  MoveL 4571 to (30.32, 60.2, -219.61) mm, rotated rx -167.81 ry 3.47 rz -52.11 deg; joints [-1.862, -33.382, 100.556, 145.163, 95.8, 28.312, -1.714]
  MoveL 4572 to (32.46, 60.06, -219.75) mm, rotated rx -167.81 ry 3.47 rz -52.11 deg; joints [-1.941, -33.35, 100.546, 145.092, 95.836, 28.324, -1.714]
  MoveL 4573 to (34.58, 59.96, -219.77) mm, rotated rx -167.81 ry 3.47 rz -52.11 deg; joints [-2.017, -33.309, 100.528, 145.023, 95.871, 28.336, -1.714]
  MoveL 4574 to (35.08, 59.57, -220.44) mm, rotated rx -167.81 ry 3.47 rz -52.11 deg; joints [-2.042, -33.346, 100.585, 144.999, 95.893, 28.332, -1.714]
  MoveL 4575 to (34.76, 59.5, -220.77) mm, rotated rx -167.81 ry 3.47 rz -52.11 deg; joints [-2.034, -33.375, 100.611, 145.006, 95.89, 28.331, -1.714]
  MoveL 4576 to (34.71, 59.48, -220.97) mm, rotated rx -167.81 ry 3.47 rz -52.11 deg; joints [-2.035, -33.389, 100.623, 145.005, 95.888, 28.332, -1.714]
  MoveL 4577 to (34.93, 59.52, -221.07) mm, rotated rx -167.81 ry 3.47 rz -52.11 deg; joints [-2.044, -33.39, 100.622, 144.997, 95.888, 28.337, -1.714]
  MoveL 4578 to (35.33, 59.66, -221.1) mm, rotated rx -167.81 ry 3.47 rz -52.11 deg; joints [-2.059, -33.381, 100.607, 144.985, 95.886, 28.345, -1.714]
  MoveC 4579 to (36.23, 60.13, -221.1) mm, rotated rx -167.81 ry 3.47 rz -52.11 deg; joints [-2.092, -33.356, 100.556, 144.957, 95.873, 28.37, -1.714] to (37.1, 60.66, -221.1) mm, rotated rx -167.81 ry 3.47 rz -52.11 deg; joints [-2.124, -33.33, 100.502, 144.93, 95.857, 28.397, -1.714]
  MoveL 4580 to (37.1, 60.66, -221.1) mm, rotated rx -167.81 ry 3.47 rz -52.11 deg; joints [-2.124, -33.331, 100.502, 144.93, 95.856, 28.397, -1.714]
  MoveL 4581 to (37.57, 60.93, -221.12) mm, rotated rx -167.81 ry 3.47 rz -52.11 deg; joints [-2.142, -33.318, 100.475, 144.915, 95.848, 28.411, -1.714]
  MoveL 4582 to (38.04, 61.18, -221.17) mm, rotated rx -167.81 ry 3.47 rz -52.11 deg; joints [-2.16, -33.308, 100.45, 144.9, 95.84, 28.425, -1.714]
  MoveL 4583 to (38.56, 61.45, -221.24) mm, rotated rx -167.81 ry 3.47 rz -52.11 deg; joints [-2.179, -33.298, 100.425, 144.883, 95.833, 28.44, -1.714]
  MoveL 4584 to (39.08, 61.73, -221.28) mm, rotated rx -167.81 ry 3.47 rz -52.11 deg; joints [-2.199, -33.285, 100.397, 144.867, 95.824, 28.456, -1.714]
  MoveL 4585 to (40.13, 62.35, -221.3) mm, rotated rx -167.81 ry 3.47 rz -52.11 deg; joints [-2.238, -33.256, 100.333, 144.835, 95.805, 28.488, -1.714]
  MoveL 4586 to (40.62, 62.62, -221.34) mm, rotated rx -167.81 ry 3.47 rz -52.11 deg; joints [-2.256, -33.244, 100.307, 144.819, 95.797, 28.502, -1.714]
  MoveL 4587 to (41.05, 62.82, -221.41) mm, rotated rx -167.81 ry 3.47 rz -52.11 deg; joints [-2.272, -33.237, 100.288, 144.805, 95.791, 28.514, -1.714]
  MoveL 4588 to (41.45, 63, -221.5) mm, rotated rx -167.81 ry 3.47 rz -52.11 deg; joints [-2.288, -33.232, 100.272, 144.792, 95.786, 28.525, -1.714]
  MoveL 4589 to (41.83, 63.19, -221.56) mm, rotated rx -167.81 ry 3.47 rz -52.11 deg; joints [-2.303, -33.225, 100.255, 144.78, 95.78, 28.536, -1.714]
  MoveL 4590 to (42.22, 63.4, -221.6) mm, rotated rx -167.81 ry 3.47 rz -52.11 deg; joints [-2.317, -33.216, 100.234, 144.767, 95.774, 28.548, -1.714]
  MoveL 4591 to (44.46, 64.76, -221.6) mm, rotated rx -167.81 ry 3.47 rz -52.11 deg; joints [-2.399, -33.15, 100.092, 144.699, 95.731, 28.618, -1.714]
  MoveL 4592 to (47.08, 66.03, -221.94) mm, rotated rx -167.81 ry 3.47 rz -52.11 deg; joints [-2.498, -33.098, 99.968, 144.615, 95.694, 28.692, -1.714]
  MoveL 4593 to (48.31, 66.38, -222.37) mm, rotated rx -167.81 ry 3.47 rz -52.11 deg; joints [-2.548, -33.094, 99.943, 144.572, 95.688, 28.72, -1.714]
  MoveL 4594 to (49.5, 66.55, -222.98) mm, rotated rx -167.81 ry 3.47 rz -52.11 deg; joints [-2.598, -33.105, 99.942, 144.529, 95.691, 28.743, -1.714]
  MoveL 4595 to (50.63, 66.52, -223.75) mm, rotated rx -167.81 ry 3.47 rz -52.11 deg; joints [-2.648, -33.13, 99.966, 144.484, 95.701, 28.76, -1.714]
  MoveL 4596 to (51.72, 66.31, -224.7) mm, rotated rx -167.81 ry 3.47 rz -52.11 deg; joints [-2.698, -33.17, 100.014, 144.439, 95.719, 28.771, -1.714]
  MoveL 4597 to (53.75, 65.31, -227.12) mm, rotated rx -167.81 ry 3.47 rz -52.11 deg; joints [-2.799, -33.293, 100.184, 144.347, 95.78, 28.776, -1.714]
  MoveL 4598 to (55.07, 63.94, -229.53) mm, rotated rx -167.81 ry 3.47 rz -52.11 deg; joints [-2.875, -33.436, 100.393, 144.276, 95.851, 28.762, -1.714]
  MoveL 4599 to (55.28, 63.26, -230.48) mm, rotated rx -167.81 ry 3.47 rz -52.11 deg; joints [-2.893, -33.501, 100.491, 144.257, 95.882, 28.748, -1.714]
  MoveL 4600 to (55.19, 62.59, -231.25) mm, rotated rx -167.81 ry 3.47 rz -52.11 deg; joints [-2.899, -33.561, 100.584, 144.25, 95.91, 28.731, -1.714]
  MoveL 4601 to (55.03, 62.26, -231.58) mm, rotated rx -167.81 ry 3.47 rz -52.11 deg; joints [-2.897, -33.59, 100.629, 144.251, 95.923, 28.72, -1.714]
  MoveL 4602 to (54.8, 61.92, -231.86) mm, rotated rx -167.81 ry 3.47 rz -52.11 deg; joints [-2.892, -33.617, 100.673, 144.255, 95.936, 28.709, -1.714]
  MoveL 4603 to (54.11, 61.26, -232.29) mm, rotated rx -167.81 ry 3.47 rz -52.11 deg; joints [-2.871, -33.668, 100.758, 144.271, 95.958, 28.683, -1.714]
  MoveL 4604 to (53.11, 60.6, -232.55) mm, rotated rx -167.81 ry 3.47 rz -52.11 deg; joints [-2.838, -33.715, 100.838, 144.298, 95.978, 28.652, -1.714]
  MoveL 4605 to (51.82, 59.94, -232.63) mm, rotated rx -167.81 ry 3.47 rz -52.11 deg; joints [-2.792, -33.757, 100.915, 144.337, 95.995, 28.618, -1.714]
  MoveL 4606 to (51.34, 59.73, -232.63) mm, rotated rx -167.81 ry 3.47 rz -52.11 deg; joints [-2.775, -33.77, 100.939, 144.352, 96, 28.606, -1.714]
  MoveL 4607 to (50.92, 59.56, -232.6) mm, rotated rx -167.81 ry 3.47 rz -52.11 deg; joints [-2.759, -33.779, 100.957, 144.365, 96.004, 28.596, -1.714]
  MoveL 4608 to (50.53, 59.42, -232.55) mm, rotated rx -167.81 ry 3.47 rz -52.11 deg; joints [-2.744, -33.786, 100.971, 144.378, 96.007, 28.586, -1.714]
  MoveL 4609 to (50.14, 59.29, -232.48) mm, rotated rx -167.81 ry 3.47 rz -52.11 deg; joints [-2.729, -33.792, 100.984, 144.391, 96.009, 28.578, -1.714]
  MoveL 4610 to (49.72, 59.14, -232.43) mm, rotated rx -167.81 ry 3.47 rz -52.11 deg; joints [-2.714, -33.8, 101, 144.404, 96.012, 28.568, -1.714]
  MoveL 4611 to (49.26, 58.94, -232.41) mm, rotated rx -167.81 ry 3.47 rz -52.11 deg; joints [-2.696, -33.811, 101.021, 144.419, 96.017, 28.556, -1.714]
  MoveL 4612 to (44.04, 56.58, -232.4) mm, rotated rx -167.81 ry 3.47 rz -52.11 deg; joints [-2.506, -33.953, 101.285, 144.581, 96.072, 28.425, -1.714]
  MoveL 4613 to (43.33, 56.28, -232.39) mm, rotated rx -167.81 ry 3.47 rz -52.11 deg; joints [-2.48, -33.971, 101.318, 144.603, 96.079, 28.408, -1.714]
  MoveL 4614 to (42.72, 56.05, -232.38) mm, rotated rx -167.81 ry 3.47 rz -52.11 deg; joints [-2.457, -33.987, 101.345, 144.622, 96.083, 28.395, -1.714]
  MoveL 4615 to (42.16, 55.93, -232.37) mm, rotated rx -167.81 ry 3.47 rz -52.11 deg; joints [-2.437, -34, 101.362, 144.64, 96.082, 28.386, -1.714]
  MoveL 4616 to (41.62, 55.89, -232.33) mm, rotated rx -167.81 ry 3.47 rz -52.11 deg; joints [-2.417, -34.009, 101.371, 144.658, 96.077, 28.38, -1.714]
  MoveL 4617 to (41.29, 55.92, -232.17) mm, rotated rx -167.81 ry 3.47 rz -52.11 deg; joints [-2.403, -34.005, 101.365, 144.67, 96.072, 28.377, -1.714]
  MoveL 4618 to (41.29, 55.95, -231.86) mm, rotated rx -167.81 ry 3.47 rz -52.11 deg; joints [-2.399, -33.985, 101.348, 144.673, 96.074, 28.374, -1.714]
  MoveL 4619 to (41.65, 55.96, -231.37) mm, rotated rx -167.81 ry 3.47 rz -52.11 deg; joints [-2.407, -33.947, 101.319, 144.667, 96.083, 28.371, -1.714]
  MoveL 4620 to (41.42, 56.54, -230.4) mm, rotated rx -167.81 ry 3.47 rz -52.11 deg; joints [-2.387, -33.883, 101.228, 144.685, 96.057, 28.38, -1.714]
  MoveL 4621 to (39.59, 56.9, -230.1) mm, rotated rx -167.81 ry 3.47 rz -52.11 deg; joints [-2.318, -33.897, 101.21, 144.749, 96.015, 28.377, -1.714]
  MoveL 4622 to (37.66, 57.25, -229.89) mm, rotated rx -167.81 ry 3.47 rz -52.11 deg; joints [-2.246, -33.919, 101.196, 144.815, 95.971, 28.374, -1.714]
  MoveL 4623 to (35.56, 57.62, -229.77) mm, rotated rx -167.81 ry 3.47 rz -52.11 deg; joints [-2.17, -33.948, 101.188, 144.885, 95.922, 28.372, -1.714]
  MoveL 4624 to (31.35, 58.33, -229.77) mm, rotated rx -167.81 ry 3.47 rz -52.11 deg; joints [-2.019, -34.024, 101.185, 145.024, 95.824, 28.37, -1.714]
  MoveL 4625 to (29.4, 58.66, -229.68) mm, rotated rx -167.81 ry 3.47 rz -52.11 deg; joints [-1.948, -34.054, 101.179, 145.089, 95.779, 28.367, -1.714]
  MoveL 4626 to (27.29, 59.01, -229.68) mm, rotated rx -167.81 ry 3.47 rz -52.11 deg; joints [-1.873, -34.092, 101.177, 145.158, 95.73, 28.366, -1.714]
  MoveL 4627 to (25.18, 59.46, -229.68) mm, rotated rx -167.81 ry 3.47 rz -52.11 deg; joints [-1.797, -34.128, 101.166, 145.228, 95.675, 28.369, -1.714]
  MoveL 4628 to (22.7, 60.03, -229.5) mm, rotated rx -167.81 ry 3.47 rz -52.11 deg; joints [-1.707, -34.158, 101.142, 145.312, 95.609, 28.371, -1.714]
  MoveL 4629 to (20.49, 60.27, -229.27) mm, rotated rx -167.81 ry 3.47 rz -52.11 deg; joints [-1.625, -34.185, 101.138, 145.386, 95.566, 28.362, -1.714]
  MoveL 4630 to (18.33, 60.54, -229.15) mm, rotated rx -167.81 ry 3.47 rz -52.11 deg; joints [-1.546, -34.217, 101.137, 145.458, 95.521, 28.355, -1.714]
  MoveL 4631 to (16.23, 60.89, -229.04) mm, rotated rx -167.81 ry 3.47 rz -52.11 deg; joints [-1.469, -34.247, 101.128, 145.528, 95.472, 28.352, -1.714]
  MoveL 4632 to (14.12, 61.23, -228.82) mm, rotated rx -167.81 ry 3.47 rz -52.11 deg; joints [-1.392, -34.271, 101.115, 145.599, 95.424, 28.348, -1.714]
  MoveL 4633 to (12.02, 61.58, -228.72) mm, rotated rx -167.81 ry 3.47 rz -52.11 deg; joints [-1.315, -34.301, 101.106, 145.669, 95.375, 28.345, -1.714]
  MoveL 4634 to (9.91, 61.92, -228.61) mm, rotated rx -167.81 ry 3.47 rz -52.11 deg; joints [-1.239, -34.331, 101.097, 145.739, 95.326, 28.342, -1.714]
  MoveL 4635 to (7.8, 62.25, -228.39) mm, rotated rx -167.81 ry 3.47 rz -52.11 deg; joints [-1.161, -34.354, 101.084, 145.81, 95.278, 28.338, -1.714]
  MoveL 4636 to (5.7, 62.59, -228.29) mm, rotated rx -167.81 ry 3.47 rz -52.11 deg; joints [-1.085, -34.384, 101.075, 145.88, 95.229, 28.335, -1.714]
  MoveL 4637 to (3.59, 62.93, -228.18) mm, rotated rx -167.81 ry 3.47 rz -52.11 deg; joints [-1.008, -34.414, 101.065, 145.95, 95.18, 28.332, -1.714]
  MoveL 4638 to (1.48, 63.24, -227.98) mm, rotated rx -167.81 ry 3.47 rz -52.11 deg; joints [-0.93, -34.438, 101.053, 146.021, 95.132, 28.326, -1.714]
  MoveL 4639 to (-0.63, 63.58, -227.88) mm, rotated rx -167.81 ry 3.47 rz -52.11 deg; joints [-0.854, -34.468, 101.044, 146.091, 95.083, 28.323, -1.714]
  MoveL 4640 to (-2.46, 63.79, -227.62) mm, rotated rx -167.81 ry 3.47 rz -52.11 deg; joints [-0.785, -34.485, 101.033, 146.153, 95.045, 28.315, -1.714]
  MoveL 4641 to (-4.13, 63.93, -227.25) mm, rotated rx -167.81 ry 3.47 rz -52.11 deg; joints [-0.721, -34.492, 101.022, 146.211, 95.016, 28.304, -1.714]
  MoveL 4642 to (-5.65, 63.98, -226.75) mm, rotated rx -167.81 ry 3.47 rz -52.11 deg; joints [-0.661, -34.49, 101.01, 146.265, 94.994, 28.29, -1.714]
  MoveL 4643 to (-4.6, 63.55, -225.91) mm, rotated rx -167.81 ry 3.47 rz -52.11 deg; joints [-0.688, -34.423, 100.994, 146.239, 95.042, 28.27, -1.714]
  MoveL 4644 to (-4.93, 63.61, -225.88) mm, rotated rx -167.81 ry 3.47 rz -52.11 deg; joints [-0.676, -34.427, 100.991, 146.25, 95.034, 28.27, -1.714]
  MoveL 4645 to (-5.24, 63.69, -225.83) mm, rotated rx -167.81 ry 3.47 rz -52.11 deg; joints [-0.664, -34.429, 100.985, 146.26, 95.025, 28.271, -1.714]
  MoveL 4646 to (-5.56, 63.87, -225.78) mm, rotated rx -167.81 ry 3.47 rz -52.11 deg; joints [-0.652, -34.429, 100.972, 146.272, 95.011, 28.274, -1.714]
  MoveL 4647 to (-5.9, 64.11, -225.74) mm, rotated rx -167.81 ry 3.47 rz -52.11 deg; joints [-0.64, -34.43, 100.954, 146.283, 94.993, 28.28, -1.714]
  MoveL 4648 to (-6.28, 64.42, -225.72) mm, rotated rx -167.81 ry 3.47 rz -52.11 deg; joints [-0.627, -34.431, 100.932, 146.296, 94.971, 28.289, -1.714]
  MoveL 4649 to (-9.71, 67.65, -225.72) mm, rotated rx -167.81 ry 3.47 rz -52.11 deg; joints [-0.511, -34.447, 100.701, 146.41, 94.74, 28.388, -1.714]
  MoveL 4650 to (-10.01, 67.91, -225.69) mm, rotated rx -167.81 ry 3.47 rz -52.11 deg; joints [-0.501, -34.447, 100.682, 146.421, 94.721, 28.395, -1.714]
  MoveL 4651 to (-10.39, 68.27, -225.69) mm, rotated rx -167.81 ry 3.47 rz -52.11 deg; joints [-0.488, -34.449, 100.656, 146.433, 94.695, 28.406, -1.714]
  MoveL 4652 to (-11.16, 68.96, -225.65) mm, rotated rx -167.81 ry 3.47 rz -52.11 deg; joints [-0.461, -34.45, 100.605, 146.459, 94.646, 28.426, -1.714]
  MoveL 4653 to (-13.06, 70.76, -225.65) mm, rotated rx -167.81 ry 3.47 rz -52.11 deg; joints [-0.397, -34.459, 100.476, 146.522, 94.517, 28.48, -1.714]
  MoveL 4654 to (-13.85, 71.42, -225.63) mm, rotated rx -167.81 ry 3.47 rz -52.11 deg; joints [-0.371, -34.462, 100.429, 146.548, 94.468, 28.5, -1.714]
  MoveL 4655 to (-14.92, 72.4, -225.7) mm, rotated rx -167.81 ry 3.47 rz -52.11 deg; joints [-0.336, -34.471, 100.361, 146.582, 94.397, 28.53, -1.714]
  MoveL 4656 to (-15.68, 73.29, -225.95) mm, rotated rx -167.81 ry 3.47 rz -52.11 deg; joints [-0.314, -34.487, 100.307, 146.605, 94.333, 28.561, -1.714]
  MoveL 4657 to (-16.13, 74.1, -226.39) mm, rotated rx -167.81 ry 3.47 rz -52.11 deg; joints [-0.304, -34.51, 100.266, 146.616, 94.277, 28.593, -1.714]
  MoveL 4658 to (-16.25, 74.47, -226.68) mm, rotated rx -167.81 ry 3.47 rz -52.11 deg; joints [-0.305, -34.525, 100.25, 146.617, 94.252, 28.61, -1.714]
  MoveL 4659 to (-16.28, 74.82, -227.02) mm, rotated rx -167.81 ry 3.47 rz -52.11 deg; joints [-0.308, -34.541, 100.237, 146.615, 94.229, 28.627, -1.714]
  MoveL 4660 to (-16.13, 75.46, -227.83) mm, rotated rx -167.81 ry 3.47 rz -52.11 deg; joints [-0.324, -34.578, 100.221, 146.602, 94.188, 28.662, -1.714]
  MoveL 4661 to (-15.68, 76.02, -228.83) mm, rotated rx -167.81 ry 3.47 rz -52.11 deg; joints [-0.354, -34.623, 100.219, 146.578, 94.155, 28.698, -1.714]
  MoveL 4662 to (-13.85, 76.87, -231.39) mm, rotated rx -167.81 ry 3.47 rz -52.11 deg; joints [-0.451, -34.733, 100.251, 146.496, 94.112, 28.775, -1.714]
  MoveL 4663 to (-11.47, 77.17, -233.95) mm, rotated rx -167.81 ry 3.47 rz -52.11 deg; joints [-0.567, -34.843, 100.324, 146.395, 94.109, 28.835, -1.714]
  MoveL 4664 to (-9.19, 76.69, -235.78) mm, rotated rx -167.81 ry 3.47 rz -52.11 deg; joints [-0.668, -34.921, 100.428, 146.303, 94.153, 28.857, -1.714]
  MoveL 4665 to (-8.08, 76.15, -236.42) mm, rotated rx -167.81 ry 3.47 rz -52.11 deg; joints [-0.714, -34.948, 100.491, 146.261, 94.193, 28.852, -1.714]
  MoveL 4666 to (-7, 75.42, -236.88) mm, rotated rx -167.81 ry 3.47 rz -52.11 deg; joints [-0.757, -34.968, 100.562, 146.222, 94.246, 28.838, -1.714]
  MoveL 4667 to (-4.92, 73.38, -237.25) mm, rotated rx -167.81 ry 3.47 rz -52.11 deg; joints [-0.831, -34.984, 100.727, 146.149, 94.387, 28.781, -1.714]
  MoveL 4668 to (-2.9, 70.96, -237.25) mm, rotated rx -167.81 ry 3.47 rz -52.11 deg; joints [-0.899, -34.983, 100.905, 146.082, 94.55, 28.704, -1.714]
  MoveL 4669 to (-2.23, 70.2, -237.26) mm, rotated rx -167.81 ry 3.47 rz -52.11 deg; joints [-0.921, -34.983, 100.962, 146.059, 94.603, 28.68, -1.714]
  MoveL 4670 to (-1.56, 69.4, -237.26) mm, rotated rx -167.81 ry 3.47 rz -52.11 deg; joints [-0.944, -34.983, 101.021, 146.037, 94.657, 28.654, -1.714]
  MoveL 4671 to (-1.24, 69.02, -237.27) mm, rotated rx -167.81 ry 3.47 rz -52.11 deg; joints [-0.955, -34.983, 101.049, 146.026, 94.683, 28.642, -1.714]
  MoveL 4672 to (-0.8, 68.52, -237.3) mm, rotated rx -167.81 ry 3.47 rz -52.11 deg; joints [-0.969, -34.984, 101.087, 146.011, 94.716, 28.627, -1.714]
  MoveL 4673 to (-0.4, 68.08, -237.35) mm, rotated rx -167.81 ry 3.47 rz -52.11 deg; joints [-0.984, -34.987, 101.121, 145.997, 94.746, 28.613, -1.714]
  MoveL 4674 to (-0.04, 67.72, -237.43) mm, rotated rx -167.81 ry 3.47 rz -52.11 deg; joints [-0.997, -34.99, 101.15, 145.984, 94.77, 28.603, -1.714]
  MoveL 4675 to (0.28, 67.39, -237.48) mm, rotated rx -167.81 ry 3.47 rz -52.11 deg; joints [-1.008, -34.992, 101.177, 145.973, 94.793, 28.594, -1.714]
  MoveL 4676 to (0.6, 67.04, -237.51) mm, rotated rx -167.81 ry 3.47 rz -52.11 deg; joints [-1.019, -34.993, 101.203, 145.962, 94.816, 28.583, -1.714]
  MoveL 4677 to (1.6, 65.84, -237.51) mm, rotated rx -167.81 ry 3.47 rz -52.11 deg; joints [-1.053, -34.992, 101.291, 145.928, 94.898, 28.545, -1.714]
  MoveL 4678 to (1.94, 65.47, -237.53) mm, rotated rx -167.81 ry 3.47 rz -52.11 deg; joints [-1.065, -34.992, 101.319, 145.916, 94.923, 28.533, -1.714]
  MoveL 4679 to (2.25, 65.16, -237.55) mm, rotated rx -167.81 ry 3.47 rz -52.11 deg; joints [-1.076, -34.993, 101.342, 145.905, 94.945, 28.524, -1.714]
  MoveL 4680 to (2.55, 64.91, -237.6) mm, rotated rx -167.81 ry 3.47 rz -52.11 deg; joints [-1.086, -34.994, 101.361, 145.895, 94.962, 28.517, -1.714]
  MoveL 4681 to (2.81, 64.76, -237.67) mm, rotated rx -167.81 ry 3.47 rz -52.11 deg; joints [-1.096, -34.995, 101.373, 145.885, 94.974, 28.514, -1.714]
  MoveL 4682 to (3.07, 64.67, -237.74) mm, rotated rx -167.81 ry 3.47 rz -52.11 deg; joints [-1.106, -34.996, 101.381, 145.876, 94.982, 28.513, -1.714]
  MoveL 4683 to (1.89, 65.73, -238.54) mm, rotated rx -167.81 ry 3.47 rz -52.11 deg; joints [-1.075, -35.053, 101.345, 145.908, 94.898, 28.555, -1.714]
  MoveL 4684 to (3.57, 65.19, -238.94) mm, rotated rx -167.81 ry 3.47 rz -52.11 deg; joints [-1.14, -35.053, 101.39, 145.849, 94.949, 28.552, -1.714]
  MoveL 4685 to (5.37, 64.66, -239.21) mm, rotated rx -167.81 ry 3.47 rz -52.11 deg; joints [-1.207, -35.042, 101.426, 145.787, 95.003, 28.548, -1.714]
  MoveL 4686 to (7.29, 64.11, -239.39) mm, rotated rx -167.81 ry 3.47 rz -52.11 deg; joints [-1.277, -35.024, 101.458, 145.722, 95.06, 28.543, -1.714]
  MoveL 4687 to (9.35, 63.55, -239.58) mm, rotated rx -167.81 ry 3.47 rz -52.11 deg; joints [-1.353, -35.004, 101.49, 145.653, 95.12, 28.538, -1.714]
  MoveL 4688 to (11.4, 62.96, -239.68) mm, rotated rx -167.81 ry 3.47 rz -52.11 deg; joints [-1.427, -34.978, 101.519, 145.584, 95.182, 28.532, -1.714]
  MoveL 4689 to (13.46, 62.38, -239.78) mm, rotated rx -167.81 ry 3.47 rz -52.11 deg; joints [-1.501, -34.952, 101.548, 145.515, 95.244, 28.525, -1.714]
  MoveL 4690 to (15.51, 61.8, -239.97) mm, rotated rx -167.81 ry 3.47 rz -52.11 deg; joints [-1.576, -34.932, 101.58, 145.446, 95.304, 28.52, -1.714]
  MoveL 4691 to (17.56, 61.21, -240.07) mm, rotated rx -167.81 ry 3.47 rz -52.11 deg; joints [-1.651, -34.906, 101.609, 145.377, 95.366, 28.513, -1.714]
  MoveL 4692 to (19.61, 60.62, -240.17) mm, rotated rx -167.81 ry 3.47 rz -52.11 deg; joints [-1.725, -34.88, 101.637, 145.308, 95.428, 28.506, -1.714]
  MoveL 4693 to (21.66, 60.04, -240.37) mm, rotated rx -167.81 ry 3.47 rz -52.11 deg; joints [-1.8, -34.859, 101.67, 145.238, 95.488, 28.501, -1.714]
  MoveL 4694 to (25.76, 58.84, -240.58) mm, rotated rx -167.81 ry 3.47 rz -52.11 deg; joints [-1.949, -34.807, 101.726, 145.1, 95.611, 28.486, -1.714]
  MoveL 4695 to (27.48, 58.34, -240.78) mm, rotated rx -167.81 ry 3.47 rz -52.11 deg; joints [-2.013, -34.792, 101.755, 145.041, 95.661, 28.481, -1.714]
  MoveL 4696 to (29.38, 57.83, -240.86) mm, rotated rx -167.81 ry 3.47 rz -52.11 deg; joints [-2.082, -34.766, 101.777, 144.977, 95.716, 28.476, -1.714]
  MoveL 4697 to (31.38, 57.35, -240.87) mm, rotated rx -167.81 ry 3.47 rz -52.11 deg; joints [-2.153, -34.733, 101.791, 144.911, 95.771, 28.472, -1.714]
  MoveL 4698 to (33.94, 56.59, -240.98) mm, rotated rx -167.81 ry 3.47 rz -52.11 deg; joints [-2.246, -34.698, 101.825, 144.824, 95.847, 28.462, -1.714]
  MoveL 4699 to (36.37, 55.75, -241.07) mm, rotated rx -167.81 ry 3.47 rz -52.11 deg; joints [-2.334, -34.666, 101.866, 144.741, 95.927, 28.447, -1.714]
  MoveL 4700 to (38.48, 55.08, -241.17) mm, rotated rx -167.81 ry 3.47 rz -52.11 deg; joints [-2.411, -34.638, 101.897, 144.67, 95.992, 28.438, -1.714]
  MoveL 4701 to (40.44, 54.49, -241.34) mm, rotated rx -167.81 ry 3.47 rz -52.11 deg; joints [-2.483, -34.617, 101.927, 144.602, 96.05, 28.431, -1.714]
  MoveL 4702 to (42.26, 53.92, -241.62) mm, rotated rx -167.81 ry 3.47 rz -52.11 deg; joints [-2.552, -34.605, 101.962, 144.538, 96.103, 28.425, -1.714]
  MoveL 4703 to (44.07, 53.35, -241.91) mm, rotated rx -167.81 ry 3.47 rz -52.11 deg; joints [-2.62, -34.593, 101.997, 144.475, 96.157, 28.419, -1.714]
  MoveL 4704 to (45.85, 52.76, -242.2) mm, rotated rx -167.81 ry 3.47 rz -52.11 deg; joints [-2.688, -34.583, 102.035, 144.412, 96.211, 28.412, -1.714]
  MoveL 4705 to (47.75, 52.16, -242.35) mm, rotated rx -167.81 ry 3.47 rz -52.11 deg; joints [-2.758, -34.562, 102.064, 144.346, 96.268, 28.405, -1.714]
  MoveL 4706 to (48.07, 51.59, -242.98) mm, rotated rx -167.81 ry 3.47 rz -52.11 deg; joints [-2.776, -34.602, 102.135, 144.327, 96.297, 28.392, -1.714]
  MoveL 4707 to (47.76, 51.54, -243.28) mm, rotated rx -167.81 ry 3.47 rz -52.11 deg; joints [-2.769, -34.629, 102.159, 144.334, 96.292, 28.392, -1.714]
  MoveL 4708 to (47.74, 51.49, -243.48) mm, rotated rx -167.81 ry 3.47 rz -52.11 deg; joints [-2.77, -34.642, 102.171, 144.333, 96.292, 28.393, -1.714]
  MoveL 4709 to (47.99, 51.48, -243.57) mm, rotated rx -167.81 ry 3.47 rz -52.11 deg; joints [-2.781, -34.643, 102.174, 144.324, 96.296, 28.395, -1.714]
  MoveL 4710 to (48.43, 51.53, -243.59) mm, rotated rx -167.81 ry 3.47 rz -52.11 deg; joints [-2.797, -34.634, 102.165, 144.309, 96.299, 28.4, -1.714]
  MoveL 4711 to (48.91, 51.62, -243.6) mm, rotated rx -167.81 ry 3.47 rz -52.11 deg; joints [-2.814, -34.623, 102.15, 144.294, 96.301, 28.408, -1.714]
  MoveL 4712 to (49.84, 51.91, -243.63) mm, rotated rx -167.81 ry 3.47 rz -52.11 deg; joints [-2.849, -34.601, 102.115, 144.264, 96.298, 28.426, -1.714]
  MoveL 4713 to (51.34, 52.38, -243.63) mm, rotated rx -167.81 ry 3.47 rz -52.11 deg; joints [-2.904, -34.563, 102.056, 144.217, 96.293, 28.456, -1.714]
  MoveL 4714 to (52.28, 52.65, -243.65) mm, rotated rx -167.81 ry 3.47 rz -52.11 deg; joints [-2.938, -34.54, 102.022, 144.187, 96.291, 28.473, -1.714]
  MoveL 4715 to (53.28, 52.96, -243.65) mm, rotated rx -167.81 ry 3.47 rz -52.11 deg; joints [-2.974, -34.515, 101.983, 144.155, 96.288, 28.493, -1.714]
  MoveL 4716 to (53.78, 53.11, -243.66) mm, rotated rx -167.81 ry 3.47 rz -52.11 deg; joints [-2.993, -34.503, 101.964, 144.14, 96.287, 28.503, -1.714]
  MoveL 4717 to (54.23, 53.24, -243.69) mm, rotated rx -167.81 ry 3.47 rz -52.11 deg; joints [-3.01, -34.494, 101.949, 144.125, 96.285, 28.511, -1.714]
  MoveL 4718 to (54.66, 53.35, -243.74) mm, rotated rx -167.81 ry 3.47 rz -52.11 deg; joints [-3.026, -34.486, 101.936, 144.111, 96.285, 28.519, -1.714]
  MoveL 4719 to (55.05, 53.45, -243.8) mm, rotated rx -167.81 ry 3.47 rz -52.11 deg; joints [-3.041, -34.48, 101.925, 144.098, 96.284, 28.527, -1.714]
  MoveL 4720 to (55.46, 53.55, -243.85) mm, rotated rx -167.81 ry 3.47 rz -52.11 deg; joints [-3.056, -34.474, 101.914, 144.085, 96.284, 28.535, -1.714]
  MoveL 4721 to (55.9, 53.67, -243.89) mm, rotated rx -167.81 ry 3.47 rz -52.11 deg; joints [-3.073, -34.464, 101.899, 144.07, 96.283, 28.543, -1.714]
  MoveL 4722 to (56.36, 53.8, -243.91) mm, rotated rx -167.81 ry 3.47 rz -52.11 deg; joints [-3.09, -34.454, 101.883, 144.055, 96.282, 28.552, -1.714]
  MoveL 4723 to (56.78, 53.9, -243.95) mm, rotated rx -167.81 ry 3.47 rz -52.11 deg; joints [-3.106, -34.447, 101.871, 144.042, 96.282, 28.56, -1.714]
  MoveL 4724 to (57.18, 53.99, -244.01) mm, rotated rx -167.81 ry 3.47 rz -52.11 deg; joints [-3.121, -34.441, 101.861, 144.028, 96.282, 28.567, -1.714]
  MoveL 4725 to (57.58, 54.08, -244.06) mm, rotated rx -167.81 ry 3.47 rz -52.11 deg; joints [-3.136, -34.434, 101.85, 144.015, 96.282, 28.574, -1.714]
  MoveL 4726 to (58.01, 54.19, -244.1) mm, rotated rx -167.81 ry 3.47 rz -52.11 deg; joints [-3.152, -34.426, 101.836, 144.001, 96.282, 28.582, -1.714]
  MoveL 4727 to (58.5, 54.35, -244.1) mm, rotated rx -167.81 ry 3.47 rz -52.11 deg; joints [-3.17, -34.413, 101.816, 143.986, 96.28, 28.592, -1.714]
  MoveL 4728 to (61.35, 54.98, -244.45) mm, rotated rx -167.81 ry 3.47 rz -52.11 deg; joints [-3.277, -34.366, 101.74, 143.892, 96.281, 28.643, -1.714]
  MoveL 4729 to (62.64, 55.06, -244.9) mm, rotated rx -167.81 ry 3.47 rz -52.11 deg; joints [-3.329, -34.365, 101.736, 143.846, 96.29, 28.661, -1.714]
  MoveL 4730 to (63.83, 54.97, -245.52) mm, rotated rx -167.81 ry 3.47 rz -52.11 deg; joints [-3.38, -34.38, 101.754, 143.801, 96.304, 28.675, -1.714]
  MoveL 4731 to (65.95, 54.31, -247.3) mm, rotated rx -167.81 ry 3.47 rz -52.11 deg; joints [-3.479, -34.455, 101.859, 143.711, 96.351, 28.688, -1.714]
  MoveL 4732 to (67.71, 53.01, -249.8) mm, rotated rx -167.81 ry 3.47 rz -52.11 deg; joints [-3.573, -34.591, 102.055, 143.624, 96.42, 28.682, -1.714]
  MoveL 4733 to (68.7, 51.51, -252.29) mm, rotated rx -167.81 ry 3.47 rz -52.11 deg; joints [-3.639, -34.747, 102.277, 143.56, 96.488, 28.662, -1.714]
  MoveL 4734 to (68.76, 50.85, -253.27) mm, rotated rx -167.81 ry 3.47 rz -52.11 deg; joints [-3.653, -34.816, 102.375, 143.546, 96.514, 28.65, -1.714]
  MoveL 4735 to (68.52, 50.26, -254.07) mm, rotated rx -167.81 ry 3.47 rz -52.11 deg; joints [-3.654, -34.88, 102.463, 143.543, 96.535, 28.635, -1.714]
  MoveL 4736 to (68.29, 49.99, -254.4) mm, rotated rx -167.81 ry 3.47 rz -52.11 deg; joints [-3.65, -34.91, 102.504, 143.546, 96.543, 28.627, -1.714]
  MoveL 4737 to (67.99, 49.73, -254.69) mm, rotated rx -167.81 ry 3.47 rz -52.11 deg; joints [-3.643, -34.938, 102.543, 143.552, 96.549, 28.619, -1.714]
  MoveL 4738 to (67.16, 49.27, -255.14) mm, rotated rx -167.81 ry 3.47 rz -52.11 deg; joints [-3.618, -34.99, 102.613, 143.573, 96.559, 28.6, -1.714]
  MoveL 4739 to (66.04, 48.87, -255.4) mm, rotated rx -167.81 ry 3.47 rz -52.11 deg; joints [-3.581, -35.036, 102.675, 143.605, 96.562, 28.58, -1.714]
  MoveL 4740 to (64.63, 48.53, -255.49) mm, rotated rx -167.81 ry 3.47 rz -52.11 deg; joints [-3.531, -35.077, 102.727, 143.649, 96.561, 28.557, -1.714]
  MoveL 4741 to (62.06, 48.03, -255.49) mm, rotated rx -167.81 ry 3.47 rz -52.11 deg; joints [-3.437, -35.139, 102.805, 143.731, 96.553, 28.519, -1.714]
  MoveL 4742 to (61.63, 47.96, -255.46) mm, rotated rx -167.81 ry 3.47 rz -52.11 deg; joints [-3.421, -35.147, 102.816, 143.745, 96.551, 28.512, -1.714]
  MoveL 4743 to (61.23, 47.91, -255.41) mm, rotated rx -167.81 ry 3.47 rz -52.11 deg; joints [-3.406, -35.153, 102.824, 143.758, 96.549, 28.507, -1.714]
  MoveL 4744 to (60.84, 47.87, -255.35) mm, rotated rx -167.81 ry 3.47 rz -52.11 deg; joints [-3.391, -35.158, 102.83, 143.772, 96.546, 28.501, -1.714]
  MoveL 4745 to (60.42, 47.81, -255.3) mm, rotated rx -167.81 ry 3.47 rz -52.11 deg; joints [-3.375, -35.165, 102.838, 143.786, 96.544, 28.495, -1.714]
  MoveL 4746 to (59.92, 47.73, -255.26) mm, rotated rx -167.81 ry 3.47 rz -52.11 deg; joints [-3.356, -35.174, 102.85, 143.802, 96.542, 28.488, -1.714]
  MoveL 4747 to (59.4, 47.66, -255.2) mm, rotated rx -167.81 ry 3.47 rz -52.11 deg; joints [-3.336, -35.182, 102.86, 143.819, 96.539, 28.481, -1.714]
  MoveL 4748 to (58.87, 47.57, -255.18) mm, rotated rx -167.81 ry 3.47 rz -52.11 deg; joints [-3.317, -35.194, 102.875, 143.837, 96.537, 28.473, -1.714]
  MoveL 4749 to (58.24, 47.44, -255.2) mm, rotated rx -167.81 ry 3.47 rz -52.11 deg; joints [-3.294, -35.21, 102.895, 143.857, 96.535, 28.464, -1.714]
  MoveL 4750 to (57.39, 47.25, -255.27) mm, rotated rx -167.81 ry 3.47 rz -52.11 deg; joints [-3.264, -35.235, 102.926, 143.883, 96.533, 28.451, -1.714]
  MoveL 4751 to (56.88, 47.15, -255.27) mm, rotated rx -167.81 ry 3.47 rz -52.11 deg; joints [-3.245, -35.247, 102.941, 143.9, 96.532, 28.443, -1.714]
  MoveL 4752 to (56.39, 47.05, -255.26) mm, rotated rx -167.81 ry 3.47 rz -52.11 deg; joints [-3.227, -35.259, 102.956, 143.915, 96.53, 28.436, -1.714]
  MoveL 4753 to (55.93, 46.97, -255.24) mm, rotated rx -167.81 ry 3.47 rz -52.11 deg; joints [-3.21, -35.268, 102.968, 143.931, 96.528, 28.429, -1.714]
  MoveL 4754 to (55.52, 46.92, -255.19) mm, rotated rx -167.81 ry 3.47 rz -52.11 deg; joints [-3.194, -35.274, 102.975, 143.944, 96.526, 28.423, -1.714]
  MoveL 4755 to (55.12, 46.89, -255.13) mm, rotated rx -167.81 ry 3.47 rz -52.11 deg; joints [-3.179, -35.28, 102.981, 143.958, 96.523, 28.419, -1.714]
  MoveL 4756 to (54.7, 46.9, -255.08) mm, rotated rx -167.81 ry 3.47 rz -52.11 deg; joints [-3.163, -35.285, 102.984, 143.972, 96.517, 28.415, -1.714]
  MoveL 4757 to (54.29, 46.95, -255.02) mm, rotated rx -167.81 ry 3.47 rz -52.11 deg; joints [-3.148, -35.29, 102.983, 143.986, 96.509, 28.414, -1.714]
  MoveL 4758 to (54.08, 47.04, -254.86) mm, rotated rx -167.81 ry 3.47 rz -52.11 deg; joints [-3.138, -35.283, 102.971, 143.995, 96.503, 28.413, -1.714]
  MoveL 4759 to (54.18, 47.1, -254.54) mm, rotated rx -167.81 ry 3.47 rz -52.11 deg; joints [-3.138, -35.26, 102.951, 143.995, 96.505, 28.412, -1.714]
  MoveL 4760 to (54.61, 47.11, -254.05) mm, rotated rx -167.81 ry 3.47 rz -52.11 deg; joints [-3.148, -35.22, 102.92, 143.986, 96.515, 28.409, -1.714]
  MoveL 4761 to (53.78, 47.42, -253.2) mm, rotated rx -167.81 ry 3.47 rz -52.11 deg; joints [-3.107, -35.18, 102.868, 144.023, 96.496, 28.404, -1.714]
  MoveL 4762 to (49.85, 49.08, -253.2) mm, rotated rx -167.81 ry 3.47 rz -52.11 deg; joints [-2.965, -35.24, 102.79, 144.158, 96.353, 28.441, -1.714]
  MoveL 4763 to (48.01, 49.85, -253.13) mm, rotated rx -167.81 ry 3.47 rz -52.11 deg; joints [-2.898, -35.263, 102.749, 144.222, 96.286, 28.458, -1.714]
  MoveL 4764 to (46.17, 50.64, -252.99) mm, rotated rx -167.81 ry 3.47 rz -52.11 deg; joints [-2.83, -35.281, 102.704, 144.286, 96.219, 28.474, -1.714]
  MoveL 4765 to (44.07, 51.55, -252.79) mm, rotated rx -167.81 ry 3.47 rz -52.11 deg; joints [-2.753, -35.3, 102.65, 144.36, 96.143, 28.492, -1.714]
  MoveL 4766 to (42.07, 52.41, -252.58) mm, rotated rx -167.81 ry 3.47 rz -52.11 deg; joints [-2.678, -35.316, 102.598, 144.431, 96.071, 28.509, -1.714]
  MoveL 4767 to (40.06, 53.26, -252.47) mm, rotated rx -167.81 ry 3.47 rz -52.11 deg; joints [-2.605, -35.339, 102.551, 144.5, 95.997, 28.526, -1.714]
  MoveL 4768 to (38.09, 54.08, -252.47) mm, rotated rx -167.81 ry 3.47 rz -52.11 deg; joints [-2.534, -35.367, 102.51, 144.567, 95.925, 28.545, -1.714]
  MoveL 4769 to (36.26, 54.85, -252.41) mm, rotated rx -167.81 ry 3.47 rz -52.11 deg; joints [-2.468, -35.39, 102.469, 144.63, 95.858, 28.561, -1.714]
  MoveL 4770 to (34.53, 55.57, -252.29) mm, rotated rx -167.81 ry 3.47 rz -52.11 deg; joints [-2.405, -35.408, 102.427, 144.689, 95.795, 28.575, -1.714]
  MoveL 4771 to (32.65, 56.36, -252.23) mm, rotated rx -167.81 ry 3.47 rz -52.11 deg; joints [-2.337, -35.431, 102.384, 144.754, 95.726, 28.591, -1.714]
  MoveL 4772 to (30.68, 57.18, -252.04) mm, rotated rx -167.81 ry 3.47 rz -52.11 deg; joints [-2.264, -35.448, 102.334, 144.822, 95.654, 28.607, -1.714]
  MoveL 4773 to (26.74, 58.82, -251.86) mm, rotated rx -167.81 ry 3.47 rz -52.11 deg; joints [-2.121, -35.492, 102.241, 144.956, 95.51, 28.64, -1.714]
  MoveL 4774 to (24.77, 59.64, -251.68) mm, rotated rx -167.81 ry 3.47 rz -52.11 deg; joints [-2.049, -35.509, 102.191, 145.024, 95.438, 28.655, -1.714]
  MoveL 4775 to (22.79, 60.45, -251.5) mm, rotated rx -167.81 ry 3.47 rz -52.11 deg; joints [-1.977, -35.526, 102.14, 145.092, 95.367, 28.67, -1.714]
  MoveL 4776 to (20.82, 61.27, -251.5) mm, rotated rx -167.81 ry 3.47 rz -52.11 deg; joints [-1.907, -35.553, 102.097, 145.158, 95.293, 28.688, -1.714]
  MoveL 4777 to (18.85, 62.08, -251.33) mm, rotated rx -167.81 ry 3.47 rz -52.11 deg; joints [-1.834, -35.57, 102.046, 145.226, 95.222, 28.703, -1.714]
  MoveL 4778 to (16.87, 62.88, -251.15) mm, rotated rx -167.81 ry 3.47 rz -52.11 deg; joints [-1.762, -35.586, 101.996, 145.294, 95.15, 28.717, -1.714]
  MoveL 4779 to (14.9, 63.7, -251.15) mm, rotated rx -167.81 ry 3.47 rz -52.11 deg; joints [-1.692, -35.613, 101.952, 145.359, 95.076, 28.735, -1.714]
  MoveL 4780 to (13.08, 64.39, -250.95) mm, rotated rx -167.81 ry 3.47 rz -52.11 deg; joints [-1.625, -35.627, 101.908, 145.421, 95.013, 28.745, -1.714]
  MoveL 4781 to (11.45, 64.93, -250.63) mm, rotated rx -167.81 ry 3.47 rz -52.11 deg; joints [-1.563, -35.631, 101.867, 145.478, 94.962, 28.75, -1.714]
  MoveL 4782 to (9.98, 65.33, -250.17) mm, rotated rx -167.81 ry 3.47 rz -52.11 deg; joints [-1.505, -35.625, 101.83, 145.531, 94.922, 28.749, -1.714]
  MoveL 4783 to (10.77, 64.81, -249.41) mm, rotated rx -167.81 ry 3.47 rz -52.11 deg; joints [-1.524, -35.57, 101.828, 145.512, 94.971, 28.725, -1.714]
  MoveL 4784 to (10.41, 65.01, -249.4) mm, rotated rx -167.81 ry 3.47 rz -52.11 deg; joints [-1.511, -35.573, 101.815, 145.524, 94.954, 28.73, -1.714]
  MoveC 4785 to (8.21, 67.81, -249.4) mm, rotated rx -167.81 ry 3.47 rz -52.11 deg; joints [-1.437, -35.573, 101.61, 145.6, 94.769, 28.821, -1.714] to (6.26, 70.79, -249.4) mm, rotated rx -167.81 ry 3.47 rz -52.11 deg; joints [-1.372, -35.564, 101.387, 145.667, 94.577, 28.92, -1.714]
  MoveL 4786 to (6.26, 70.79, -249.4) mm, rotated rx -167.81 ry 3.47 rz -52.11 deg; joints [-1.372, -35.564, 101.387, 145.667, 94.577, 28.92, -1.714]
  MoveL 4787 to (6, 71.17, -249.38) mm, rotated rx -167.81 ry 3.47 rz -52.11 deg; joints [-1.363, -35.561, 101.357, 145.677, 94.552, 28.933, -1.714]
  MoveL 4788 to (5.74, 71.51, -249.32) mm, rotated rx -167.81 ry 3.47 rz -52.11 deg; joints [-1.353, -35.558, 101.33, 145.686, 94.531, 28.943, -1.714]
  MoveL 4789 to (5.49, 71.83, -249.26) mm, rotated rx -167.81 ry 3.47 rz -52.11 deg; joints [-1.344, -35.554, 101.303, 145.695, 94.51, 28.952, -1.714]
  MoveL 4790 to (5.23, 72.18, -249.22) mm, rotated rx -167.81 ry 3.47 rz -52.11 deg; joints [-1.335, -35.55, 101.275, 145.704, 94.487, 28.963, -1.714]
  MoveL 4791 to (4.95, 72.56, -249.19) mm, rotated rx -167.81 ry 3.47 rz -52.11 deg; joints [-1.326, -35.548, 101.245, 145.714, 94.462, 28.976, -1.714]
  MoveL 4792 to (4.66, 72.99, -249.17) mm, rotated rx -167.81 ry 3.47 rz -52.11 deg; joints [-1.316, -35.546, 101.212, 145.724, 94.435, 28.99, -1.714]
  MoveL 4793 to (4.08, 73.87, -249.17) mm, rotated rx -167.81 ry 3.47 rz -52.11 deg; joints [-1.297, -35.543, 101.146, 145.744, 94.378, 29.019, -1.714]
  MoveL 4794 to (3.33, 75.11, -249.27) mm, rotated rx -167.81 ry 3.47 rz -52.11 deg; joints [-1.273, -35.543, 101.055, 145.768, 94.298, 29.062, -1.714]
  MoveL 4795 to (2.82, 76.2, -249.54) mm, rotated rx -167.81 ry 3.47 rz -52.11 deg; joints [-1.26, -35.552, 100.983, 145.783, 94.228, 29.103, -1.714]
  MoveL 4796 to (2.55, 77.13, -250) mm, rotated rx -167.81 ry 3.47 rz -52.11 deg; joints [-1.257, -35.57, 100.93, 145.788, 94.168, 29.142, -1.714]
  MoveL 4797 to (2.52, 77.9, -250.64) mm, rotated rx -167.81 ry 3.47 rz -52.11 deg; joints [-1.265, -35.598, 100.896, 145.784, 94.119, 29.18, -1.714]
  MoveL 4798 to (2.74, 78.51, -251.46) mm, rotated rx -167.81 ry 3.47 rz -52.11 deg; joints [-1.284, -35.634, 100.881, 145.77, 94.08, 29.216, -1.714]
  MoveL 4799 to (3.19, 78.96, -252.47) mm, rotated rx -167.81 ry 3.47 rz -52.11 deg; joints [-1.313, -35.68, 100.884, 145.746, 94.052, 29.25, -1.714]
  MoveL 4800 to (4.83, 79.39, -255.02) mm, rotated rx -167.81 ry 3.47 rz -52.11 deg; joints [-1.403, -35.8, 100.948, 145.668, 94.027, 29.313, -1.714]
  MoveL 4801 to (6.86, 79.14, -257.58) mm, rotated rx -167.81 ry 3.47 rz -52.11 deg; joints [-1.506, -35.923, 101.064, 145.578, 94.045, 29.353, -1.714]
  MoveL 4802 to (7.82, 78.73, -258.59) mm, rotated rx -167.81 ry 3.47 rz -52.11 deg; joints [-1.552, -35.973, 101.132, 145.537, 94.071, 29.358, -1.714]
  MoveL 4803 to (8.73, 78.15, -259.41) mm, rotated rx -167.81 ry 3.47 rz -52.11 deg; joints [-1.593, -36.016, 101.208, 145.499, 94.108, 29.354, -1.714]
  MoveL 4804 to (9.6, 77.38, -260.05) mm, rotated rx -167.81 ry 3.47 rz -52.11 deg; joints [-1.631, -36.052, 101.291, 145.464, 94.156, 29.34, -1.714]
  MoveL 4805 to (10.43, 76.43, -260.51) mm, rotated rx -167.81 ry 3.47 rz -52.11 deg; joints [-1.664, -36.08, 101.382, 145.431, 94.216, 29.316, -1.714]
  MoveL 4806 to (11.97, 73.97, -260.88) mm, rotated rx -167.81 ry 3.47 rz -52.11 deg; joints [-1.72, -36.113, 101.584, 145.375, 94.369, 29.238, -1.714]
  MoveL 4807 to (12.45, 73.04, -260.88) mm, rotated rx -167.81 ry 3.47 rz -52.11 deg; joints [-1.736, -36.119, 101.656, 145.358, 94.426, 29.206, -1.714]
  MoveL 4808 to (12.69, 72.57, -260.88) mm, rotated rx -167.81 ry 3.47 rz -52.11 deg; joints [-1.744, -36.122, 101.692, 145.35, 94.455, 29.19, -1.714]
  MoveL 4809 to (12.92, 72.16, -260.91) mm, rotated rx -167.81 ry 3.47 rz -52.11 deg; joints [-1.752, -36.125, 101.725, 145.341, 94.481, 29.177, -1.714]
  MoveL 4810 to (13.14, 71.79, -260.96) mm, rotated rx -167.81 ry 3.47 rz -52.11 deg; joints [-1.76, -36.13, 101.755, 145.333, 94.504, 29.165, -1.714]
  MoveL 4811 to (13.35, 71.45, -261.01) mm, rotated rx -167.81 ry 3.47 rz -52.11 deg; joints [-1.767, -36.135, 101.783, 145.325, 94.525, 29.154, -1.714]
  MoveL 4812 to (13.56, 71.09, -261.06) mm, rotated rx -167.81 ry 3.47 rz -52.11 deg; joints [-1.775, -36.14, 101.812, 145.317, 94.547, 29.143, -1.714]
  MoveL 4813 to (13.79, 70.68, -261.08) mm, rotated rx -167.81 ry 3.47 rz -52.11 deg; joints [-1.783, -36.143, 101.845, 145.309, 94.573, 29.129, -1.714]
  MoveL 4814 to (14.02, 70.24, -261.09) mm, rotated rx -167.81 ry 3.47 rz -52.11 deg; joints [-1.79, -36.146, 101.879, 145.301, 94.6, 29.114, -1.714]
  MoveL 4815 to (14.27, 69.74, -261.08) mm, rotated rx -167.81 ry 3.47 rz -52.11 deg; joints [-1.799, -36.149, 101.916, 145.292, 94.631, 29.096, -1.714]
  MoveL 4816 to (14.51, 69.27, -261.09) mm, rotated rx -167.81 ry 3.47 rz -52.11 deg; joints [-1.807, -36.152, 101.953, 145.283, 94.66, 29.08, -1.714]
  MoveL 4817 to (14.75, 68.84, -261.11) mm, rotated rx -167.81 ry 3.47 rz -52.11 deg; joints [-1.815, -36.156, 101.987, 145.275, 94.686, 29.066, -1.714]
  MoveL 4818 to (14.98, 68.43, -261.16) mm, rotated rx -167.81 ry 3.47 rz -52.11 deg; joints [-1.823, -36.161, 102.02, 145.266, 94.712, 29.052, -1.714]
  MoveL 4819 to (15.25, 68, -261.23) mm, rotated rx -167.81 ry 3.47 rz -52.11 deg; joints [-1.833, -36.167, 102.056, 145.256, 94.738, 29.039, -1.714]
  MoveL 4820 to (15.56, 67.48, -261.3) mm, rotated rx -167.81 ry 3.47 rz -52.11 deg; joints [-1.844, -36.173, 102.098, 145.244, 94.77, 29.022, -1.714]
  MoveL 4821 to (15.83, 66.97, -261.31) mm, rotated rx -167.81 ry 3.47 rz -52.11 deg; joints [-1.854, -36.177, 102.137, 145.235, 94.802, 29.005, -1.714]
  MoveL 4822 to (16.07, 66.51, -261.32) mm, rotated rx -167.81 ry 3.47 rz -52.11 deg; joints [-1.862, -36.179, 102.172, 145.226, 94.83, 28.989, -1.714]
  MoveL 4823 to (16.31, 66.04, -261.32) mm, rotated rx -167.81 ry 3.47 rz -52.11 deg; joints [-1.87, -36.182, 102.208, 145.217, 94.859, 28.973, -1.714]
  MoveL 4824 to (16.63, 65.46, -261.33) mm, rotated rx -167.81 ry 3.47 rz -52.11 deg; joints [-1.88, -36.185, 102.252, 145.206, 94.895, 28.953, -1.714]
  MoveL 4825 to (16.93, 64.96, -261.34) mm, rotated rx -167.81 ry 3.47 rz -52.11 deg; joints [-1.891, -36.188, 102.29, 145.195, 94.927, 28.936, -1.714]
  MoveL 4826 to (17.21, 64.54, -261.34) mm, rotated rx -167.81 ry 3.47 rz -52.11 deg; joints [-1.9, -36.189, 102.322, 145.185, 94.954, 28.922, -1.714]
  MoveL 4827 to (17.45, 64.29, -261.35) mm, rotated rx -167.81 ry 3.47 rz -52.11 deg; joints [-1.908, -36.189, 102.34, 145.177, 94.971, 28.914, -1.714]
  MoveL 4828 to (17.66, 64.12, -261.35) mm, rotated rx -167.81 ry 3.47 rz -52.11 deg; joints [-1.916, -36.187, 102.351, 145.169, 94.983, 28.909, -1.714]
  MoveL 4829 to (16.91, 64.69, -261.94) mm, rotated rx -167.81 ry 3.47 rz -52.11 deg; joints [-1.897, -36.23, 102.34, 145.189, 94.934, 28.934, -1.714]
  MoveL 4830 to (18.18, 64.3, -262.47) mm, rotated rx -167.81 ry 3.47 rz -52.11 deg; joints [-1.949, -36.243, 102.381, 145.142, 94.969, 28.935, -1.714]
  MoveL 4831 to (19.63, 63.7, -262.85) mm, rotated rx -167.81 ry 3.47 rz -52.11 deg; joints [-2.005, -36.247, 102.43, 145.09, 95.019, 28.928, -1.714]
  MoveL 4832 to (21.29, 62.9, -263.11) mm, rotated rx -167.81 ry 3.47 rz -52.11 deg; joints [-2.067, -36.242, 102.488, 145.031, 95.085, 28.912, -1.714]
  MoveL 4833 to (23.1, 61.93, -263.23) mm, rotated rx -167.81 ry 3.47 rz -52.11 deg; joints [-2.133, -36.229, 102.551, 144.969, 95.163, 28.89, -1.714]
  MoveL 4834 to (24.95, 60.93, -263.33) mm, rotated rx -167.81 ry 3.47 rz -52.11 deg; joints [-2.199, -36.212, 102.615, 144.906, 95.244, 28.866, -1.714]
  MoveL 4835 to (28.7, 58.88, -263.5) mm, rotated rx -167.81 ry 3.47 rz -52.11 deg; joints [-2.335, -36.178, 102.744, 144.777, 95.408, 28.816, -1.714]
  MoveL 4836 to (30.57, 57.86, -263.68) mm, rotated rx -167.81 ry 3.47 rz -52.11 deg; joints [-2.404, -36.167, 102.811, 144.712, 95.489, 28.792, -1.714]
  MoveL 4837 to (34.31, 55.8, -263.86) mm, rotated rx -167.81 ry 3.47 rz -52.11 deg; joints [-2.539, -36.132, 102.939, 144.582, 95.653, 28.741, -1.714]
  MoveL 4838 to (36.18, 54.77, -264.05) mm, rotated rx -167.81 ry 3.47 rz -52.11 deg; joints [-2.608, -36.12, 103.007, 144.516, 95.734, 28.717, -1.714]
  MoveL 4839 to (38.04, 53.74, -264.14) mm, rotated rx -167.81 ry 3.47 rz -52.11 deg; joints [-2.676, -36.102, 103.071, 144.451, 95.815, 28.691, -1.714]
  MoveL 4840 to (39.76, 52.76, -264.35) mm, rotated rx -167.81 ry 3.47 rz -52.11 deg; joints [-2.74, -36.094, 103.137, 144.39, 95.89, 28.668, -1.714]
  MoveL 4841 to (41.82, 51.63, -264.5) mm, rotated rx -167.81 ry 3.47 rz -52.11 deg; joints [-2.816, -36.077, 103.209, 144.317, 95.979, 28.641, -1.714]
  MoveL 4842 to (44.07, 50.39, -264.61) mm, rotated rx -167.81 ry 3.47 rz -52.11 deg; joints [-2.898, -36.056, 103.285, 144.238, 96.077, 28.609, -1.714]
  MoveL 4843 to (45.94, 49.35, -264.61) mm, rotated rx -167.81 ry 3.47 rz -52.11 deg; joints [-2.965, -36.031, 103.343, 144.173, 96.159, 28.582, -1.714]
  MoveL 4844 to (47.71, 48.36, -264.69) mm, rotated rx -167.81 ry 3.47 rz -52.11 deg; joints [-3.03, -36.013, 103.402, 144.111, 96.237, 28.557, -1.714]
  MoveL 4845 to (49.3, 47.45, -264.86) mm, rotated rx -167.81 ry 3.47 rz -52.11 deg; joints [-3.09, -36.003, 103.461, 144.054, 96.306, 28.535, -1.714]
  MoveL 4846 to (50.92, 46.51, -265.07) mm, rotated rx -167.81 ry 3.47 rz -52.11 deg; joints [-3.15, -35.996, 103.524, 143.995, 96.377, 28.512, -1.714]
  MoveL 4847 to (52.98, 45.36, -265.21) mm, rotated rx -167.81 ry 3.47 rz -52.11 deg; joints [-3.226, -35.977, 103.595, 143.921, 96.466, 28.483, -1.714]
  MoveL 4848 to (55.23, 44.1, -265.32) mm, rotated rx -167.81 ry 3.47 rz -52.11 deg; joints [-3.309, -35.954, 103.669, 143.841, 96.563, 28.45, -1.714]
  MoveL 4849 to (58.96, 42.04, -265.32) mm, rotated rx -167.81 ry 3.47 rz -52.11 deg; joints [-3.444, -35.903, 103.781, 143.71, 96.725, 28.395, -1.714]
  MoveL 4850 to (59.03, 41.73, -266.01) mm, rotated rx -167.81 ry 3.47 rz -52.11 deg; joints [-3.456, -35.949, 103.837, 143.699, 96.735, 28.393, -1.714]
  MoveL 4851 to (58.72, 41.76, -266.36) mm, rotated rx -167.81 ry 3.47 rz -52.11 deg; joints [-3.449, -35.977, 103.854, 143.706, 96.725, 28.397, -1.714]
  MoveL 4852 to (58.71, 41.75, -266.58) mm, rotated rx -167.81 ry 3.47 rz -52.11 deg; joints [-3.451, -35.991, 103.865, 143.704, 96.723, 28.399, -1.714]
  MoveL 4853 to (58.97, 41.7, -266.69) mm, rotated rx -167.81 ry 3.47 rz -52.11 deg; joints [-3.462, -35.993, 103.87, 143.694, 96.728, 28.401, -1.714]
  MoveL 4854 to (59.42, 41.68, -266.72) mm, rotated rx -167.81 ry 3.47 rz -52.11 deg; joints [-3.479, -35.986, 103.867, 143.679, 96.735, 28.403, -1.714]
  MoveL 4855 to (59.9, 41.69, -266.74) mm, rotated rx -167.81 ry 3.47 rz -52.11 deg; joints [-3.496, -35.977, 103.861, 143.663, 96.741, 28.407, -1.714]
  MoveL 4856 to (60.33, 41.7, -266.79) mm, rotated rx -167.81 ry 3.47 rz -52.11 deg; joints [-3.513, -35.97, 103.856, 143.648, 96.746, 28.411, -1.714]
  MoveL 4857 to (60.73, 41.7, -266.86) mm, rotated rx -167.81 ry 3.47 rz -52.11 deg; joints [-3.528, -35.966, 103.853, 143.634, 96.751, 28.415, -1.714]
  MoveL 4858 to (61.14, 41.7, -266.92) mm, rotated rx -167.81 ry 3.47 rz -52.11 deg; joints [-3.544, -35.961, 103.849, 143.62, 96.755, 28.419, -1.714]
  MoveL 4859 to (61.59, 41.72, -266.96) mm, rotated rx -167.81 ry 3.47 rz -52.11 deg; joints [-3.561, -35.953, 103.843, 143.605, 96.76, 28.424, -1.714]
  MoveL 4860 to (62.11, 41.76, -266.98) mm, rotated rx -167.81 ry 3.47 rz -52.11 deg; joints [-3.58, -35.943, 103.834, 143.588, 96.765, 28.429, -1.714]
  MoveL 4861 to (62.64, 41.77, -267.04) mm, rotated rx -167.81 ry 3.47 rz -52.11 deg; joints [-3.6, -35.936, 103.828, 143.57, 96.771, 28.434, -1.714]
  MoveL 4862 to (63.16, 41.8, -267.08) mm, rotated rx -167.81 ry 3.47 rz -52.11 deg; joints [-3.62, -35.926, 103.819, 143.552, 96.776, 28.44, -1.714]
  MoveL 4863 to (63.68, 41.84, -267.08) mm, rotated rx -167.81 ry 3.47 rz -52.11 deg; joints [-3.639, -35.915, 103.808, 143.535, 96.781, 28.445, -1.714]
  MoveL 4864 to (64.2, 41.88, -267.08) mm, rotated rx -167.81 ry 3.47 rz -52.11 deg; joints [-3.658, -35.903, 103.797, 143.518, 96.786, 28.45, -1.714]
  MoveL 4865 to (64.89, 41.96, -267.05) mm, rotated rx -167.81 ry 3.47 rz -52.11 deg; joints [-3.683, -35.885, 103.779, 143.496, 96.791, 28.458, -1.714]
  MoveL 4866 to (65.55, 42.03, -267.02) mm, rotated rx -167.81 ry 3.47 rz -52.11 deg; joints [-3.706, -35.868, 103.763, 143.475, 96.797, 28.465, -1.714]
  MoveL 4867 to (66.14, 42.08, -267.01) mm, rotated rx -167.81 ry 3.47 rz -52.11 deg; joints [-3.728, -35.854, 103.749, 143.456, 96.802, 28.471, -1.714]
  MoveL 4868 to (66.61, 42.1, -267.05) mm, rotated rx -167.81 ry 3.47 rz -52.11 deg; joints [-3.746, -35.846, 103.742, 143.44, 96.807, 28.476, -1.714]
  MoveL 4869 to (67.03, 42.11, -267.11) mm, rotated rx -167.81 ry 3.47 rz -52.11 deg; joints [-3.762, -35.84, 103.738, 143.426, 96.812, 28.48, -1.714]
  MoveL 4870 to (67.43, 42.12, -267.16) mm, rotated rx -167.81 ry 3.47 rz -52.11 deg; joints [-3.777, -35.835, 103.734, 143.412, 96.816, 28.484, -1.714]
  MoveL 4871 to (67.88, 42.14, -267.2) mm, rotated rx -167.81 ry 3.47 rz -52.11 deg; joints [-3.794, -35.827, 103.727, 143.397, 96.821, 28.488, -1.714]
  MoveL 4872 to (69.44, 42.27, -267.2) mm, rotated rx -167.81 ry 3.47 rz -52.11 deg; joints [-3.851, -35.792, 103.693, 143.346, 96.835, 28.505, -1.714]
  MoveL 4873 to (72.33, 42.29, -267.57) mm, rotated rx -167.81 ry 3.47 rz -52.11 deg; joints [-3.961, -35.752, 103.665, 143.247, 96.868, 28.532, -1.714]
  MoveL 4874 to (73.57, 42.11, -268.04) mm, rotated rx -167.81 ry 3.47 rz -52.11 deg; joints [-4.012, -35.757, 103.682, 143.2, 96.889, 28.54, -1.714]
  MoveL 4875 to (74.67, 41.8, -268.7) mm, rotated rx -167.81 ry 3.47 rz -52.11 deg; joints [-4.061, -35.779, 103.719, 143.156, 96.913, 28.545, -1.714]
  MoveL 4876 to (75.64, 41.37, -269.55) mm, rotated rx -167.81 ry 3.47 rz -52.11 deg; joints [-4.107, -35.816, 103.777, 143.114, 96.94, 28.547, -1.714]
  MoveL 4877 to (76.47, 40.81, -270.59) mm, rotated rx -167.81 ry 3.47 rz -52.11 deg; joints [-4.151, -35.871, 103.856, 143.073, 96.969, 28.545, -1.714]
  MoveL 4878 to (77.72, 39.32, -273.22) mm, rotated rx -167.81 ry 3.47 rz -52.11 deg; joints [-4.23, -36.029, 104.074, 142.998, 97.035, 28.532, -1.714]
  MoveL 4879 to (78.18, 37.79, -275.86) mm, rotated rx -167.81 ry 3.47 rz -52.11 deg; joints [-4.28, -36.204, 104.307, 142.949, 97.092, 28.513, -1.714]
  MoveL 4880 to (78.02, 37.2, -276.9) mm, rotated rx -167.81 ry 3.47 rz -52.11 deg; joints [-4.288, -36.28, 104.403, 142.941, 97.109, 28.503, -1.714]
  MoveL 4881 to (77.6, 36.72, -277.74) mm, rotated rx -167.81 ry 3.47 rz -52.11 deg; joints [-4.283, -36.349, 104.485, 142.944, 97.12, 28.493, -1.714]
  MoveL 4882 to (76.92, 36.36, -278.4) mm, rotated rx -167.81 ry 3.47 rz -52.11 deg; joints [-4.267, -36.41, 104.555, 142.958, 97.122, 28.483, -1.714]
  MoveL 4883 to (75.98, 36.1, -278.87) mm, rotated rx -167.81 ry 3.47 rz -52.11 deg; joints [-4.239, -36.464, 104.61, 142.983, 97.118, 28.474, -1.714]
  MoveL 4884 to (74.78, 35.96, -279.16) mm, rotated rx -167.81 ry 3.47 rz -52.11 deg; joints [-4.198, -36.51, 104.653, 143.019, 97.106, 28.464, -1.714]
  MoveL 4885 to (73.32, 35.93, -279.25) mm, rotated rx -167.81 ry 3.47 rz -52.11 deg; joints [-4.146, -36.548, 104.682, 143.066, 97.087, 28.454, -1.714]
  MoveL 4886 to (72.8, 35.94, -279.25) mm, rotated rx -167.81 ry 3.47 rz -52.11 deg; joints [-4.127, -36.559, 104.689, 143.084, 97.079, 28.45, -1.714]
  MoveL 4887 to (72.33, 35.95, -279.23) mm, rotated rx -167.81 ry 3.47 rz -52.11 deg; joints [-4.109, -36.568, 104.694, 143.099, 97.072, 28.447, -1.714]
  MoveL 4888 to (71.93, 35.99, -279.18) mm, rotated rx -167.81 ry 3.47 rz -52.11 deg; joints [-4.094, -36.573, 104.695, 143.113, 97.066, 28.445, -1.714]
  MoveL 4889 to (71.54, 36.02, -279.13) mm, rotated rx -167.81 ry 3.47 rz -52.11 deg; joints [-4.079, -36.577, 104.696, 143.127, 97.059, 28.443, -1.714]
  MoveL 4890 to (71.11, 36.05, -279.09) mm, rotated rx -167.81 ry 3.47 rz -52.11 deg; joints [-4.062, -36.584, 104.698, 143.142, 97.052, 28.441, -1.714]
  MoveL 4891 to (70.62, 36.07, -279.06) mm, rotated rx -167.81 ry 3.47 rz -52.11 deg; joints [-4.044, -36.593, 104.703, 143.159, 97.045, 28.438, -1.714]
  MoveL 4892 to (70.09, 36.08, -279.06) mm, rotated rx -167.81 ry 3.47 rz -52.11 deg; joints [-4.025, -36.604, 104.71, 143.176, 97.037, 28.434, -1.714]
  MoveL 4893 to (69.63, 36.1, -279.04) mm, rotated rx -167.81 ry 3.47 rz -52.11 deg; joints [-4.008, -36.613, 104.715, 143.192, 97.03, 28.431, -1.714]
  MoveL 4894 to (69.22, 36.12, -278.99) mm, rotated rx -167.81 ry 3.47 rz -52.11 deg; joints [-3.992, -36.618, 104.717, 143.206, 97.024, 28.429, -1.714]
  MoveL 4895 to (68.83, 36.15, -278.92) mm, rotated rx -167.81 ry 3.47 rz -52.11 deg; joints [-3.977, -36.622, 104.718, 143.22, 97.018, 28.426, -1.714]
  MoveL 4896 to (68.4, 36.17, -278.88) mm, rotated rx -167.81 ry 3.47 rz -52.11 deg; joints [-3.961, -36.628, 104.72, 143.234, 97.012, 28.423, -1.714]
  MoveL 4897 to (67.91, 36.19, -278.85) mm, rotated rx -167.81 ry 3.47 rz -52.11 deg; joints [-3.942, -36.637, 104.725, 143.251, 97.004, 28.42, -1.714]
  MoveL 4898 to (67.39, 36.2, -278.85) mm, rotated rx -167.81 ry 3.47 rz -52.11 deg; joints [-3.923, -36.648, 104.732, 143.269, 96.997, 28.417, -1.714]
  MoveL 4899 to (66.41, 36.29, -278.83) mm, rotated rx -167.81 ry 3.47 rz -52.11 deg; joints [-3.887, -36.667, 104.739, 143.302, 96.979, 28.413, -1.714]
  MoveC 4900 to (65.04, 36.45, -278.83) mm, rotated rx -167.81 ry 3.47 rz -52.11 deg; joints [-3.836, -36.695, 104.746, 143.348, 96.951, 28.41, -1.714] to (63.66, 36.44, -278.83) mm, rotated rx -167.81 ry 3.47 rz -52.11 deg; joints [-3.786, -36.725, 104.767, 143.394, 96.933, 28.401, -1.714]
  MoveL 4901 to (63.66, 36.44, -278.82) mm, rotated rx -167.81 ry 3.47 rz -52.11 deg; joints [-3.786, -36.724, 104.767, 143.394, 96.933, 28.4, -1.714]
  MoveL 4902 to (63, 36.49, -278.81) mm, rotated rx -167.81 ry 3.47 rz -52.11 deg; joints [-3.761, -36.737, 104.771, 143.416, 96.921, 28.398, -1.714]
  MoveL 4903 to (62.43, 36.6, -278.78) mm, rotated rx -167.81 ry 3.47 rz -52.11 deg; joints [-3.74, -36.746, 104.77, 143.436, 96.908, 28.398, -1.714]
  MoveL 4904 to (62.16, 36.72, -278.68) mm, rotated rx -167.81 ry 3.47 rz -52.11 deg; joints [-3.729, -36.744, 104.76, 143.447, 96.899, 28.399, -1.714]
  MoveL 4905 to (62.21, 36.75, -278.49) mm, rotated rx -167.81 ry 3.47 rz -52.11 deg; joints [-3.728, -36.73, 104.748, 143.447, 96.901, 28.398, -1.714]
  MoveL 4906 to (62.63, 36.67, -278.18) mm, rotated rx -167.81 ry 3.47 rz -52.11 deg; joints [-3.74, -36.703, 104.735, 143.436, 96.914, 28.393, -1.714]
  MoveL 4907 to (62.9, 36.94, -277.56) mm, rotated rx -167.81 ry 3.47 rz -52.11 deg; joints [-3.742, -36.655, 104.682, 143.434, 96.911, 28.396, -1.714]
  MoveL 4908 to (61.17, 38.01, -277.55) mm, rotated rx -167.81 ry 3.47 rz -52.11 deg; joints [-3.678, -36.677, 104.621, 143.496, 96.83, 28.427, -1.714]
  MoveL 4909 to (59.39, 39.21, -277.49) mm, rotated rx -167.81 ry 3.47 rz -52.11 deg; joints [-3.613, -36.695, 104.548, 143.561, 96.742, 28.461, -1.714]
  MoveL 4910 to (57.53, 40.52, -277.37) mm, rotated rx -167.81 ry 3.47 rz -52.11 deg; joints [-3.544, -36.708, 104.464, 143.629, 96.648, 28.499, -1.714]
  MoveL 4911 to (55.71, 41.81, -277.27) mm, rotated rx -167.81 ry 3.47 rz -52.11 deg; joints [-3.476, -36.723, 104.382, 143.696, 96.555, 28.535, -1.714]
  MoveL 4912 to (53.95, 43.05, -277.1) mm, rotated rx -167.81 ry 3.47 rz -52.11 deg; joints [-3.41, -36.732, 104.299, 143.761, 96.466, 28.57, -1.714]
  MoveL 4913 to (52.36, 44.18, -276.95) mm, rotated rx -167.81 ry 3.47 rz -52.11 deg; joints [-3.351, -36.741, 104.225, 143.819, 96.386, 28.601, -1.714]
  MoveL 4914 to (50.67, 45.36, -276.9) mm, rotated rx -167.81 ry 3.47 rz -52.11 deg; joints [-3.289, -36.757, 104.15, 143.88, 96.299, 28.635, -1.714]
  MoveL 4915 to (48.9, 46.6, -276.83) mm, rotated rx -167.81 ry 3.47 rz -52.11 deg; joints [-3.224, -36.772, 104.072, 143.944, 96.209, 28.67, -1.714]
  MoveL 4916 to (46.97, 47.95, -276.67) mm, rotated rx -167.81 ry 3.47 rz -52.11 deg; joints [-3.153, -36.783, 103.982, 144.014, 96.111, 28.707, -1.714]
  MoveL 4917 to (45.43, 49.02, -276.56) mm, rotated rx -167.81 ry 3.47 rz -52.11 deg; joints [-3.096, -36.793, 103.911, 144.069, 96.032, 28.737, -1.714]
  MoveL 4918 to (43.47, 50.39, -276.35) mm, rotated rx -167.81 ry 3.47 rz -52.11 deg; joints [-3.023, -36.801, 103.818, 144.141, 95.933, 28.774, -1.714]
  MoveL 4919 to (41.93, 51.46, -276.23) mm, rotated rx -167.81 ry 3.47 rz -52.11 deg; joints [-2.966, -36.81, 103.746, 144.196, 95.855, 28.803, -1.714]
  MoveL 4920 to (40.18, 52.67, -276.07) mm, rotated rx -167.81 ry 3.47 rz -52.11 deg; joints [-2.901, -36.818, 103.664, 144.259, 95.766, 28.836, -1.714]
  MoveL 4921 to (38.21, 54.03, -276.02) mm, rotated rx -167.81 ry 3.47 rz -52.11 deg; joints [-2.83, -36.836, 103.577, 144.328, 95.665, 28.874, -1.714]
  MoveL 4922 to (36.67, 55.1, -275.9) mm, rotated rx -167.81 ry 3.47 rz -52.11 deg; joints [-2.773, -36.845, 103.505, 144.383, 95.587, 28.903, -1.714]
  MoveL 4923 to (34.91, 56.31, -275.74) mm, rotated rx -167.81 ry 3.47 rz -52.11 deg; joints [-2.709, -36.853, 103.423, 144.446, 95.498, 28.935, -1.714]
  MoveL 4924 to (32.94, 57.66, -275.69) mm, rotated rx -167.81 ry 3.47 rz -52.11 deg; joints [-2.638, -36.87, 103.335, 144.514, 95.397, 28.973, -1.714]
  MoveL 4925 to (31.39, 58.73, -275.58) mm, rotated rx -167.81 ry 3.47 rz -52.11 deg; joints [-2.581, -36.878, 103.263, 144.569, 95.318, 29.001, -1.714]
  MoveL 4926 to (29.56, 59.98, -275.48) mm, rotated rx -167.81 ry 3.47 rz -52.11 deg; joints [-2.515, -36.89, 103.179, 144.633, 95.224, 29.035, -1.714]
  MoveL 4927 to (27.72, 61.24, -275.41) mm, rotated rx -167.81 ry 3.47 rz -52.11 deg; joints [-2.449, -36.904, 103.095, 144.696, 95.13, 29.07, -1.714]
  MoveL 4928 to (26.16, 62.28, -275.23) mm, rotated rx -167.81 ry 3.47 rz -52.11 deg; joints [-2.391, -36.908, 103.022, 144.751, 95.052, 29.096, -1.714]
  MoveL 4929 to (24.69, 63.21, -274.98) mm, rotated rx -167.81 ry 3.47 rz -52.11 deg; joints [-2.336, -36.908, 102.952, 144.804, 94.983, 29.118, -1.714]
  MoveL 4930 to (23.31, 64.06, -274.62) mm, rotated rx -167.81 ry 3.47 rz -52.11 deg; joints [-2.282, -36.9, 102.883, 144.854, 94.92, 29.135, -1.714]
  MoveL 4931 to (24.26, 62.89, -273.93) mm, rotated rx -167.81 ry 3.47 rz -52.11 deg; joints [-2.307, -36.857, 102.937, 144.827, 95.006, 29.087, -1.714]
  MoveL 4932 to (24.1, 63.05, -273.93) mm, rotated rx -167.81 ry 3.47 rz -52.11 deg; joints [-2.301, -36.857, 102.926, 144.833, 94.995, 29.092, -1.714]
  MoveL 4933 to (23.92, 63.29, -273.92) mm, rotated rx -167.81 ry 3.47 rz -52.11 deg; joints [-2.295, -36.856, 102.908, 144.84, 94.979, 29.1, -1.714]
  MoveL 4934 to (23.7, 63.69, -273.89) mm, rotated rx -167.81 ry 3.47 rz -52.11 deg; joints [-2.287, -36.852, 102.876, 144.848, 94.955, 29.113, -1.714]
  MoveL 4935 to (23.47, 64.18, -273.85) mm, rotated rx -167.81 ry 3.47 rz -52.11 deg; joints [-2.279, -36.847, 102.838, 144.857, 94.926, 29.13, -1.714]
  MoveL 4936 to (23.22, 64.74, -273.8) mm, rotated rx -167.81 ry 3.47 rz -52.11 deg; joints [-2.27, -36.84, 102.792, 144.867, 94.892, 29.149, -1.714]
  MoveL 4937 to (22.26, 67.18, -273.8) mm, rotated rx -167.81 ry 3.47 rz -52.11 deg; joints [-2.238, -36.821, 102.604, 144.903, 94.746, 29.236, -1.714]
  MoveL 4938 to (22.02, 67.74, -273.77) mm, rotated rx -167.81 ry 3.47 rz -52.11 deg; joints [-2.23, -36.814, 102.559, 144.912, 94.713, 29.255, -1.714]
  MoveL 4939 to (21.75, 68.37, -273.72) mm, rotated rx -167.81 ry 3.47 rz -52.11 deg; joints [-2.22, -36.806, 102.508, 144.923, 94.676, 29.277, -1.714]
  MoveL 4940 to (21.5, 68.94, -273.68) mm, rotated rx -167.81 ry 3.47 rz -52.11 deg; joints [-2.212, -36.8, 102.462, 144.932, 94.641, 29.297, -1.714]
  MoveL 4941 to (21.31, 69.43, -273.68) mm, rotated rx -167.81 ry 3.47 rz -52.11 deg; joints [-2.205, -36.796, 102.424, 144.939, 94.612, 29.314, -1.714]
  MoveL 4942 to (21.13, 69.89, -273.68) mm, rotated rx -167.81 ry 3.47 rz -52.11 deg; joints [-2.199, -36.791, 102.388, 144.946, 94.585, 29.33, -1.714]
  MoveL 4943 to (20.94, 70.38, -273.68) mm, rotated rx -167.81 ry 3.47 rz -52.11 deg; joints [-2.193, -36.787, 102.35, 144.953, 94.556, 29.347, -1.714]
  MoveL 4944 to (20.75, 70.85, -273.67) mm, rotated rx -167.81 ry 3.47 rz -52.11 deg; joints [-2.187, -36.783, 102.313, 144.96, 94.527, 29.364, -1.714]
  MoveL 4945 to (20.56, 71.3, -273.65) mm, rotated rx -167.81 ry 3.47 rz -52.11 deg; joints [-2.18, -36.778, 102.277, 144.967, 94.501, 29.38, -1.714]
  MoveL 4946 to (20.38, 71.72, -273.6) mm, rotated rx -167.81 ry 3.47 rz -52.11 deg; joints [-2.174, -36.771, 102.242, 144.974, 94.476, 29.394, -1.714]
  MoveL 4947 to (20.19, 72.19, -273.58) mm, rotated rx -167.81 ry 3.47 rz -52.11 deg; joints [-2.167, -36.766, 102.206, 144.981, 94.448, 29.41, -1.714]
  MoveL 4948 to (19.99, 72.68, -273.58) mm, rotated rx -167.81 ry 3.47 rz -52.11 deg; joints [-2.161, -36.762, 102.167, 144.989, 94.419, 29.427, -1.714]
  MoveL 4949 to (19.61, 73.65, -273.58) mm, rotated rx -167.81 ry 3.47 rz -52.11 deg; joints [-2.148, -36.753, 102.091, 145.002, 94.36, 29.462, -1.714]
  Set speed (1000.0 mm/s)
  MoveL 4950 to (17.73, 95.19, -273.58) mm, rotated rx -167.81 ry 3.47 rz -52.11 deg; joints [-2.11, -36.413, 100.313, 145.09, 93.173, 30.274, -1.714]
  Print: /'Flow1'
  Set speed (1000.0 mm/s)
  MoveL 4951 to (-108.71, -12.41, -72.4) mm, rotated rx -172.19 ry 6.28 rz 7.52 deg; joints [-2.84, -26.042, 88.749, 94.674, 103.86, 48.031, -36.259]
  Set speed (1000.0 mm/s)
  MoveL 4952 to (-68.04, -31.37, -72.4) mm, rotated rx -172.19 ry 6.28 rz 7.52 deg; joints [-4.191, -26.495, 90.873, 93.052, 104.574, 46.354, -36.259]
  Set speed (100.0 mm/s)
  MoveL 4953 to (-2.09, -62.13, -72.4) mm, rotated rx -172.19 ry 6.28 rz 7.52 deg; joints [-6.463, -27.055, 93.998, 90.299, 105.585, 43.727, -36.259]
  MoveL 4954 to (-1.86, -62.59, -72.4) mm, rotated rx -172.19 ry 6.28 rz 7.52 deg; joints [-6.472, -27.075, 94.045, 90.283, 105.588, 43.699, -36.259]
  MoveL 4955 to (-1.52, -63.14, -72.3) mm, rotated rx -172.19 ry 6.28 rz 7.52 deg; joints [-6.483, -27.092, 94.099, 90.262, 105.593, 43.66, -36.259]
  MoveL 4956 to (-1.22, -63.65, -72.25) mm, rotated rx -172.19 ry 6.28 rz 7.52 deg; joints [-6.493, -27.11, 94.151, 90.244, 105.597, 43.626, -36.259]
  MoveL 4957 to (-0.95, -64.15, -72.23) mm, rotated rx -172.19 ry 6.28 rz 7.52 deg; joints [-6.503, -27.13, 94.201, 90.226, 105.601, 43.594, -36.259]
  MoveL 4958 to (0.7, -67.42, -72.23) mm, rotated rx -172.19 ry 6.28 rz 7.52 deg; joints [-6.564, -27.265, 94.527, 90.116, 105.625, 43.396, -36.259]
  MoveL 4959 to (1.31, -68.74, -72.32) mm, rotated rx -172.19 ry 6.28 rz 7.52 deg; joints [-6.588, -27.324, 94.659, 90.074, 105.634, 43.321, -36.259]
  MoveL 4960 to (1.67, -69.87, -72.58) mm, rotated rx -172.19 ry 6.28 rz 7.52 deg; joints [-6.605, -27.386, 94.772, 90.044, 105.641, 43.267, -36.259]
  MoveL 4961 to (1.81, -70.81, -73.03) mm, rotated rx -172.19 ry 6.28 rz 7.52 deg; joints [-6.616, -27.449, 94.865, 90.025, 105.645, 43.235, -36.259]
  MoveL 4962 to (1.79, -71.21, -73.31) mm, rotated rx -172.19 ry 6.28 rz 7.52 deg; joints [-6.619, -27.481, 94.905, 90.02, 105.647, 43.228, -36.259]
  MoveL 4963 to (1.71, -71.55, -73.65) mm, rotated rx -172.19 ry 6.28 rz 7.52 deg; joints [-6.621, -27.514, 94.94, 90.018, 105.647, 43.225, -36.259]
  MoveL 4964 to (1.38, -72.11, -74.44) mm, rotated rx -172.19 ry 6.28 rz 7.52 deg; joints [-6.62, -27.581, 94.997, 90.022, 105.647, 43.237, -36.259]
  MoveL 4965 to (0.82, -72.47, -75.42) mm, rotated rx -172.19 ry 6.28 rz 7.52 deg; joints [-6.612, -27.651, 95.034, 90.038, 105.644, 43.27, -36.259]
  MoveL 4966 to (-1, -72.62, -77.91) mm, rotated rx -172.19 ry 6.28 rz 7.52 deg; joints [-6.578, -27.796, 95.052, 90.104, 105.631, 43.402, -36.259]
  MoveL 4967 to (-3.14, -72.05, -80.39) mm, rotated rx -172.19 ry 6.28 rz 7.52 deg; joints [-6.533, -27.909, 94.997, 90.194, 105.613, 43.577, -36.259]
  MoveL 4968 to (-4.99, -70.78, -82.16) mm, rotated rx -172.19 ry 6.28 rz 7.52 deg; joints [-6.488, -27.953, 94.872, 90.282, 105.595, 43.751, -36.259]
  MoveL 4969 to (-5.8, -69.9, -82.79) mm, rotated rx -172.19 ry 6.28 rz 7.52 deg; joints [-6.467, -27.948, 94.783, 90.325, 105.586, 43.839, -36.259]
  MoveL 4970 to (-6.53, -68.84, -83.23) mm, rotated rx -172.19 ry 6.28 rz 7.52 deg; joints [-6.445, -27.926, 94.677, 90.368, 105.577, 43.926, -36.259]
  MoveL 4971 to (-7.78, -66.2, -83.58) mm, rotated rx -172.19 ry 6.28 rz 7.52 deg; joints [-6.403, -27.83, 94.413, 90.453, 105.559, 44.1, -36.259]
  MoveL 4972 to (-8.88, -63.25, -83.59) mm, rotated rx -172.19 ry 6.28 rz 7.52 deg; joints [-6.362, -27.7, 94.116, 90.537, 105.541, 44.273, -36.259]
  MoveL 4973 to (-9.06, -62.8, -83.61) mm, rotated rx -172.19 ry 6.28 rz 7.52 deg; joints [-6.356, -27.681, 94.071, 90.551, 105.538, 44.3, -36.259]
  MoveL 4974 to (-9.24, -62.37, -83.65) mm, rotated rx -172.19 ry 6.28 rz 7.52 deg; joints [-6.349, -27.664, 94.028, 90.564, 105.535, 44.327, -36.259]
  MoveL 4975 to (-9.42, -62, -83.71) mm, rotated rx -172.19 ry 6.28 rz 7.52 deg; joints [-6.343, -27.651, 93.99, 90.576, 105.533, 44.353, -36.259]
  MoveL 4976 to (-9.61, -61.59, -83.76) mm, rotated rx -172.19 ry 6.28 rz 7.52 deg; joints [-6.337, -27.635, 93.949, 90.589, 105.53, 44.379, -36.259]
  MoveL 4977 to (-9.81, -61.09, -83.79) mm, rotated rx -172.19 ry 6.28 rz 7.52 deg; joints [-6.33, -27.614, 93.898, 90.604, 105.527, 44.41, -36.259]
  MoveL 4978 to (-10.06, -60.49, -83.82) mm, rotated rx -172.19 ry 6.28 rz 7.52 deg; joints [-6.321, -27.589, 93.838, 90.622, 105.523, 44.447, -36.259]
  MoveL 4979 to (-10.28, -59.97, -83.88) mm, rotated rx -172.19 ry 6.28 rz 7.52 deg; joints [-6.314, -27.57, 93.786, 90.638, 105.519, 44.481, -36.259]
  MoveL 4980 to (-10.48, -59.57, -83.96) mm, rotated rx -172.19 ry 6.28 rz 7.52 deg; joints [-6.307, -27.556, 93.745, 90.651, 105.517, 44.508, -36.259]
  MoveL 4981 to (-10.66, -59.17, -84.01) mm, rotated rx -172.19 ry 6.28 rz 7.52 deg; joints [-6.301, -27.541, 93.705, 90.663, 105.514, 44.534, -36.259]
  MoveL 4982 to (-10.84, -58.73, -84.03) mm, rotated rx -172.19 ry 6.28 rz 7.52 deg; joints [-6.295, -27.522, 93.66, 90.676, 105.511, 44.562, -36.259]
  MoveL 4983 to (-11.02, -58.24, -84.03) mm, rotated rx -172.19 ry 6.28 rz 7.52 deg; joints [-6.288, -27.5, 93.61, 90.69, 105.508, 44.591, -36.259]
  MoveL 4984 to (-11.21, -57.73, -84.03) mm, rotated rx -172.19 ry 6.28 rz 7.52 deg; joints [-6.281, -27.477, 93.559, 90.704, 105.505, 44.62, -36.259]
  MoveL 4985 to (-11.42, -57.2, -84.04) mm, rotated rx -172.19 ry 6.28 rz 7.52 deg; joints [-6.274, -27.454, 93.505, 90.72, 105.501, 44.652, -36.259]
  MoveL 4986 to (-11.68, -56.59, -84.07) mm, rotated rx -172.19 ry 6.28 rz 7.52 deg; joints [-6.264, -27.429, 93.443, 90.739, 105.497, 44.69, -36.259]
  MoveL 4987 to (-11.94, -56.06, -84.14) mm, rotated rx -172.19 ry 6.28 rz 7.52 deg; joints [-6.256, -27.409, 93.389, 90.756, 105.493, 44.725, -36.259]
  MoveL 4988 to (-12.17, -55.67, -84.24) mm, rotated rx -172.19 ry 6.28 rz 7.52 deg; joints [-6.249, -27.397, 93.349, 90.77, 105.49, 44.754, -36.259]
  MoveL 4989 to (-12.16, -55.66, -84.48) mm, rotated rx -172.19 ry 6.28 rz 7.52 deg; joints [-6.252, -27.407, 93.348, 90.77, 105.491, 44.765, -36.259]
  MoveL 4990 to (-11.91, -55.97, -84.84) mm, rotated rx -172.19 ry 6.28 rz 7.52 deg; joints [-6.265, -27.434, 93.379, 90.757, 105.496, 44.761, -36.259]
  MoveL 4991 to (-12.11, -56.8, -85.8) mm, rotated rx -172.19 ry 6.28 rz 7.52 deg; joints [-6.27, -27.519, 93.462, 90.753, 105.498, 44.764, -36.259]
  MoveL 4992 to (-13.84, -55.55, -85.8) mm, rotated rx -172.19 ry 6.28 rz 7.52 deg; joints [-6.209, -27.483, 93.338, 90.833, 105.472, 44.856, -36.259]
  MoveL 4993 to (-15.72, -54.23, -85.93) mm, rotated rx -172.19 ry 6.28 rz 7.52 deg; joints [-6.145, -27.452, 93.206, 90.919, 105.445, 44.959, -36.259]
  MoveL 4994 to (-17.49, -52.96, -85.99) mm, rotated rx -172.19 ry 6.28 rz 7.52 deg; joints [-6.084, -27.418, 93.08, 91.001, 105.418, 45.054, -36.259]
  MoveL 4995 to (-19.23, -51.74, -86.12) mm, rotated rx -172.19 ry 6.28 rz 7.52 deg; joints [-6.025, -27.388, 92.956, 91.08, 105.392, 45.151, -36.259]
  MoveL 4996 to (-20.98, -50.5, -86.27) mm, rotated rx -172.19 ry 6.28 rz 7.52 deg; joints [-5.965, -27.359, 92.832, 91.16, 105.365, 45.249, -36.259]
  MoveL 4997 to (-22.71, -49.27, -86.4) mm, rotated rx -172.19 ry 6.28 rz 7.52 deg; joints [-5.907, -27.328, 92.707, 91.239, 105.339, 45.346, -36.259]
  MoveL 4998 to (-24.45, -48.03, -86.6) mm, rotated rx -172.19 ry 6.28 rz 7.52 deg; joints [-5.848, -27.3, 92.582, 91.319, 105.312, 45.447, -36.259]
  MoveL 4999 to (-26.18, -46.79, -86.72) mm, rotated rx -172.19 ry 6.28 rz 7.52 deg; joints [-5.79, -27.268, 92.456, 91.397, 105.286, 45.543, -36.259]
  MoveL 5000 to (-27.92, -45.53, -86.78) mm, rotated rx -172.19 ry 6.28 rz 7.52 deg; joints [-5.73, -27.233, 92.328, 91.477, 105.258, 45.638, -36.259]
  MoveL 5001 to (-29.67, -44.27, -86.92) mm, rotated rx -172.19 ry 6.28 rz 7.52 deg; joints [-5.671, -27.201, 92.2, 91.556, 105.231, 45.738, -36.259]
  MoveL 5002 to (-31.48, -42.97, -87.1) mm, rotated rx -172.19 ry 6.28 rz 7.52 deg; joints [-5.611, -27.169, 92.066, 91.638, 105.202, 45.842, -36.259]
  MoveL 5003 to (-33.28, -41.67, -87.28) mm, rotated rx -172.19 ry 6.28 rz 7.52 deg; joints [-5.55, -27.136, 91.932, 91.72, 105.174, 45.947, -36.259]
  MoveL 5004 to (-34.8, -40.56, -87.52) mm, rotated rx -172.19 ry 6.28 rz 7.52 deg; joints [-5.501, -27.112, 91.817, 91.789, 105.15, 46.039, -36.259]
  MoveL 5005 to (-36.95, -38.99, -87.63) mm, rotated rx -172.19 ry 6.28 rz 7.52 deg; joints [-5.428, -27.068, 91.655, 91.886, 105.115, 46.16, -36.259]
  Set speed (1000.0 mm/s)
  MoveL 5006 to (-78.01, -19.85, -87.63) mm, rotated rx -172.19 ry 6.28 rz 7.52 deg; joints [-4.041, -26.651, 89.609, 93.552, 104.425, 47.813, -36.259]
  Set speed (1000.0 mm/s)
  MoveL 5007 to (-75.59, -14.65, -99.51) mm, rotated rx -172.19 ry 6.28 rz 7.52 deg; joints [-4.265, -26.815, 89.025, 93.548, 104.482, 48.592, -36.259]
  Set speed (100.0 mm/s)
  MoveL 5008 to (-49.59, -26.77, -99.51) mm, rotated rx -172.19 ry 6.28 rz 7.52 deg; joints [-5.136, -27.099, 90.344, 92.507, 104.935, 47.544, -36.259]
  MoveL 5009 to (-48.35, -27.96, -99.27) mm, rotated rx -172.19 ry 6.28 rz 7.52 deg; joints [-5.175, -27.134, 90.47, 92.448, 104.957, 47.451, -36.259]
  MoveL 5010 to (-46.87, -29.34, -99.2) mm, rotated rx -172.19 ry 6.28 rz 7.52 deg; joints [-5.225, -27.182, 90.615, 92.378, 104.983, 47.352, -36.259]
  MoveL 5011 to (-45.36, -30.74, -99.06) mm, rotated rx -172.19 ry 6.28 rz 7.52 deg; joints [-5.275, -27.229, 90.763, 92.307, 105.01, 47.248, -36.259]
  MoveL 5012 to (-43.57, -32.42, -98.92) mm, rotated rx -172.19 ry 6.28 rz 7.52 deg; joints [-5.334, -27.286, 90.941, 92.222, 105.041, 47.124, -36.259]
  MoveL 5013 to (-42, -33.87, -98.92) mm, rotated rx -172.19 ry 6.28 rz 7.52 deg; joints [-5.388, -27.339, 91.092, 92.147, 105.068, 47.023, -36.259]
  MoveL 5014 to (-40.27, -35.47, -98.76) mm, rotated rx -172.19 ry 6.28 rz 7.52 deg; joints [-5.446, -27.391, 91.259, 92.065, 105.098, 46.905, -36.259]
  MoveL 5015 to (-38.81, -36.83, -98.58) mm, rotated rx -172.19 ry 6.28 rz 7.52 deg; joints [-5.494, -27.433, 91.401, 91.995, 105.122, 46.802, -36.259]
  MoveL 5016 to (-37.31, -38.22, -98.49) mm, rotated rx -172.19 ry 6.28 rz 7.52 deg; joints [-5.544, -27.479, 91.546, 91.923, 105.148, 46.701, -36.259]
  MoveL 5017 to (-35.74, -39.66, -98.27) mm, rotated rx -172.19 ry 6.28 rz 7.52 deg; joints [-5.596, -27.523, 91.697, 91.848, 105.174, 46.591, -36.259]
  MoveL 5018 to (-34.18, -41.09, -98.11) mm, rotated rx -172.19 ry 6.28 rz 7.52 deg; joints [-5.648, -27.567, 91.845, 91.773, 105.2, 46.485, -36.259]
  MoveL 5019 to (-32.62, -42.52, -98) mm, rotated rx -172.19 ry 6.28 rz 7.52 deg; joints [-5.7, -27.613, 91.992, 91.698, 105.226, 46.381, -36.259]
  MoveL 5020 to (-31.04, -43.96, -97.83) mm, rotated rx -172.19 ry 6.28 rz 7.52 deg; joints [-5.753, -27.657, 92.14, 91.622, 105.252, 46.273, -36.259]
  MoveL 5021 to (-29.47, -45.39, -97.69) mm, rotated rx -172.19 ry 6.28 rz 7.52 deg; joints [-5.806, -27.701, 92.287, 91.547, 105.277, 46.167, -36.259]
  MoveL 5022 to (-27.86, -46.86, -97.63) mm, rotated rx -172.19 ry 6.28 rz 7.52 deg; joints [-5.861, -27.75, 92.438, 91.469, 105.303, 46.063, -36.259]
  MoveL 5023 to (-26.27, -48.28, -97.42) mm, rotated rx -172.19 ry 6.28 rz 7.52 deg; joints [-5.914, -27.791, 92.584, 91.393, 105.329, 45.954, -36.259]
  MoveL 5024 to (-24.7, -49.7, -97.29) mm, rotated rx -172.19 ry 6.28 rz 7.52 deg; joints [-5.968, -27.835, 92.728, 91.317, 105.354, 45.85, -36.259]
  MoveL 5025 to (-23.09, -51.15, -97.17) mm, rotated rx -172.19 ry 6.28 rz 7.52 deg; joints [-6.022, -27.879, 92.876, 91.239, 105.379, 45.744, -36.259]
  MoveL 5026 to (-21.69, -52.24, -96.96) mm, rotated rx -172.19 ry 6.28 rz 7.52 deg; joints [-6.069, -27.905, 92.986, 91.174, 105.401, 45.657, -36.259]
  MoveL 5027 to (-20.45, -53.03, -96.61) mm, rotated rx -172.19 ry 6.28 rz 7.52 deg; joints [-6.108, -27.912, 93.066, 91.118, 105.419, 45.581, -36.259]
  MoveL 5028 to (-19.34, -53.51, -96.08) mm, rotated rx -172.19 ry 6.28 rz 7.52 deg; joints [-6.14, -27.897, 93.115, 91.072, 105.433, 45.515, -36.259]
  MoveL 5029 to (-20.11, -52.18, -95.23) mm, rotated rx -172.19 ry 6.28 rz 7.52 deg; joints [-6.103, -27.805, 92.982, 91.117, 105.417, 45.557, -36.259]
  MoveL 5030 to (-19.65, -52.84, -95.23) mm, rotated rx -172.19 ry 6.28 rz 7.52 deg; joints [-6.119, -27.831, 93.049, 91.091, 105.424, 45.516, -36.259]
  MoveL 5031 to (-19.3, -53.45, -95.23) mm, rotated rx -172.19 ry 6.28 rz 7.52 deg; joints [-6.132, -27.857, 93.111, 91.07, 105.43, 45.478, -36.259]
  MoveL 5032 to (-19.07, -54.04, -95.22) mm, rotated rx -172.19 ry 6.28 rz 7.52 deg; joints [-6.14, -27.884, 93.171, 91.053, 105.434, 45.443, -36.259]
  MoveL 5033 to (-18.87, -54.68, -95.2) mm, rotated rx -172.19 ry 6.28 rz 7.52 deg; joints [-6.147, -27.912, 93.236, 91.036, 105.438, 45.405, -36.259]
  MoveL 5034 to (-18.66, -55.41, -95.17) mm, rotated rx -172.19 ry 6.28 rz 7.52 deg; joints [-6.155, -27.945, 93.311, 91.018, 105.442, 45.362, -36.259]
  MoveL 5035 to (-18.17, -57.45, -95.17) mm, rotated rx -172.19 ry 6.28 rz 7.52 deg; joints [-6.173, -28.042, 93.519, 90.97, 105.452, 45.247, -36.259]
  MoveL 5036 to (-18.06, -57.88, -95.15) mm, rotated rx -172.19 ry 6.28 rz 7.52 deg; joints [-6.177, -28.061, 93.563, 90.96, 105.454, 45.221, -36.259]
  MoveL 5037 to (-17.81, -58.9, -95.15) mm, rotated rx -172.19 ry 6.28 rz 7.52 deg; joints [-6.187, -28.109, 93.667, 90.936, 105.459, 45.164, -36.259]
  MoveL 5038 to (-17.69, -59.39, -95.14) mm, rotated rx -172.19 ry 6.28 rz 7.52 deg; joints [-6.191, -28.132, 93.717, 90.924, 105.461, 45.136, -36.259]
  MoveL 5039 to (-17.57, -59.86, -95.12) mm, rotated rx -172.19 ry 6.28 rz 7.52 deg; joints [-6.196, -28.154, 93.765, 90.913, 105.463, 45.108, -36.259]
  MoveL 5040 to (-17.43, -60.32, -95.09) mm, rotated rx -172.19 ry 6.28 rz 7.52 deg; joints [-6.2, -28.173, 93.811, 90.901, 105.466, 45.08, -36.259]
  MoveL 5041 to (-17.29, -60.73, -95.03) mm, rotated rx -172.19 ry 6.28 rz 7.52 deg; joints [-6.205, -28.19, 93.853, 90.89, 105.468, 45.054, -36.259]
  MoveL 5042 to (-17.16, -61.19, -95) mm, rotated rx -172.19 ry 6.28 rz 7.52 deg; joints [-6.209, -28.209, 93.899, 90.878, 105.47, 45.026, -36.259]
  MoveL 5043 to (-17.03, -61.67, -94.98) mm, rotated rx -172.19 ry 6.28 rz 7.52 deg; joints [-6.214, -28.231, 93.948, 90.867, 105.472, 44.998, -36.259]
  MoveL 5044 to (-16.91, -62.16, -94.97) mm, rotated rx -172.19 ry 6.28 rz 7.52 deg; joints [-6.219, -28.254, 93.998, 90.855, 105.475, 44.97, -36.259]
  MoveL 5045 to (-16.78, -62.63, -94.95) mm, rotated rx -172.19 ry 6.28 rz 7.52 deg; joints [-6.223, -28.275, 94.046, 90.843, 105.477, 44.942, -36.259]
  MoveL 5046 to (-16.64, -63.09, -94.92) mm, rotated rx -172.19 ry 6.28 rz 7.52 deg; joints [-6.228, -28.295, 94.093, 90.831, 105.479, 44.914, -36.259]
  MoveL 5047 to (-16.5, -63.5, -94.86) mm, rotated rx -172.19 ry 6.28 rz 7.52 deg; joints [-6.233, -28.311, 94.134, 90.82, 105.482, 44.888, -36.259]
  MoveL 5048 to (-16.35, -63.93, -94.8) mm, rotated rx -172.19 ry 6.28 rz 7.52 deg; joints [-6.238, -28.328, 94.178, 90.808, 105.484, 44.86, -36.259]
  MoveL 5049 to (-15.95, -65.32, -94.72) mm, rotated rx -172.19 ry 6.28 rz 7.52 deg; joints [-6.252, -28.388, 94.318, 90.773, 105.491, 44.778, -36.259]
  MoveL 5050 to (-15.77, -66.48, -94.85) mm, rotated rx -172.19 ry 6.28 rz 7.52 deg; joints [-6.261, -28.449, 94.435, 90.75, 105.495, 44.72, -36.259]
  MoveL 5051 to (-15.8, -67.42, -95.19) mm, rotated rx -172.19 ry 6.28 rz 7.52 deg; joints [-6.265, -28.512, 94.529, 90.737, 105.497, 44.686, -36.259]
  MoveL 5052 to (-15.9, -67.81, -95.43) mm, rotated rx -172.19 ry 6.28 rz 7.52 deg; joints [-6.265, -28.543, 94.568, 90.735, 105.497, 44.679, -36.259]
  MoveL 5053 to (-16.05, -68.15, -95.73) mm, rotated rx -172.19 ry 6.28 rz 7.52 deg; joints [-6.263, -28.575, 94.602, 90.736, 105.497, 44.677, -36.259]
  MoveL 5054 to (-16.51, -68.65, -96.49) mm, rotated rx -172.19 ry 6.28 rz 7.52 deg; joints [-6.257, -28.64, 94.652, 90.746, 105.494, 44.693, -36.259]
  MoveL 5055 to (-17.19, -68.94, -97.46) mm, rotated rx -172.19 ry 6.28 rz 7.52 deg; joints [-6.245, -28.706, 94.679, 90.768, 105.489, 44.733, -36.259]
  MoveL 5056 to (-19.21, -68.85, -100.02) mm, rotated rx -172.19 ry 6.28 rz 7.52 deg; joints [-6.206, -28.841, 94.666, 90.844, 105.471, 44.887, -36.259]
  MoveL 5057 to (-21.39, -67.99, -102.64) mm, rotated rx -172.19 ry 6.28 rz 7.52 deg; joints [-6.161, -28.942, 94.574, 90.939, 105.449, 45.086, -36.259]
  MoveL 5058 to (-22.28, -67.31, -103.66) mm, rotated rx -172.19 ry 6.28 rz 7.52 deg; joints [-6.141, -28.965, 94.504, 90.982, 105.439, 45.182, -36.259]
  MoveL 5059 to (-23.05, -66.48, -104.5) mm, rotated rx -172.19 ry 6.28 rz 7.52 deg; joints [-6.124, -28.969, 94.417, 91.023, 105.431, 45.277, -36.259]
  MoveL 5060 to (-23.68, -65.47, -105.15) mm, rotated rx -172.19 ry 6.28 rz 7.52 deg; joints [-6.109, -28.955, 94.314, 91.061, 105.423, 45.369, -36.259]
  MoveL 5061 to (-24.19, -64.31, -105.62) mm, rotated rx -172.19 ry 6.28 rz 7.52 deg; joints [-6.096, -28.923, 94.195, 91.097, 105.416, 45.459, -36.259]
  MoveL 5062 to (-24.56, -62.97, -105.9) mm, rotated rx -172.19 ry 6.28 rz 7.52 deg; joints [-6.086, -28.872, 94.059, 91.13, 105.41, 45.547, -36.259]
  MoveL 5063 to (-24.81, -61.48, -105.99) mm, rotated rx -172.19 ry 6.28 rz 7.52 deg; joints [-6.077, -28.803, 93.907, 91.161, 105.404, 45.633, -36.259]
  MoveL 5064 to (-25.16, -58.34, -106) mm, rotated rx -172.19 ry 6.28 rz 7.52 deg; joints [-6.062, -28.647, 93.587, 91.219, 105.395, 45.803, -36.259]
  MoveL 5065 to (-25.23, -57.79, -106.01) mm, rotated rx -172.19 ry 6.28 rz 7.52 deg; joints [-6.059, -28.621, 93.531, 91.23, 105.393, 45.834, -36.259]
  MoveL 5066 to (-25.33, -57.18, -106.05) mm, rotated rx -172.19 ry 6.28 rz 7.52 deg; joints [-6.056, -28.592, 93.468, 91.242, 105.391, 45.869, -36.259]
  MoveL 5067 to (-25.47, -56.43, -106.14) mm, rotated rx -172.19 ry 6.28 rz 7.52 deg; joints [-6.051, -28.56, 93.391, 91.258, 105.388, 45.915, -36.259]
  MoveL 5068 to (-25.57, -55.82, -106.18) mm, rotated rx -172.19 ry 6.28 rz 7.52 deg; joints [-6.048, -28.531, 93.329, 91.271, 105.386, 45.951, -36.259]
  MoveL 5069 to (-25.64, -55.28, -106.19) mm, rotated rx -172.19 ry 6.28 rz 7.52 deg; joints [-6.045, -28.505, 93.273, 91.281, 105.384, 45.981, -36.259]
  MoveL 5070 to (-25.7, -54.78, -106.2) mm, rotated rx -172.19 ry 6.28 rz 7.52 deg; joints [-6.043, -28.48, 93.222, 91.291, 105.382, 46.008, -36.259]
  MoveL 5071 to (-25.77, -54.32, -106.22) mm, rotated rx -172.19 ry 6.28 rz 7.52 deg; joints [-6.04, -28.459, 93.176, 91.3, 105.381, 46.034, -36.259]
  MoveL 5072 to (-26.01, -52.28, -106.23) mm, rotated rx -172.19 ry 6.28 rz 7.52 deg; joints [-6.031, -28.357, 92.966, 91.338, 105.374, 46.146, -36.259]
  MoveL 5073 to (-26.09, -51.77, -106.26) mm, rotated rx -172.19 ry 6.28 rz 7.52 deg; joints [-6.028, -28.333, 92.914, 91.349, 105.372, 46.175, -36.259]
  MoveL 5074 to (-26.18, -51.31, -106.31) mm, rotated rx -172.19 ry 6.28 rz 7.52 deg; joints [-6.025, -28.313, 92.866, 91.359, 105.37, 46.204, -36.259]
  MoveL 5075 to (-26.28, -50.86, -106.38) mm, rotated rx -172.19 ry 6.28 rz 7.52 deg; joints [-6.022, -28.294, 92.82, 91.369, 105.368, 46.232, -36.259]
  MoveL 5076 to (-26.42, -50.39, -106.44) mm, rotated rx -172.19 ry 6.28 rz 7.52 deg; joints [-6.018, -28.274, 92.771, 91.381, 105.366, 46.262, -36.259]
  MoveL 5077 to (-26.58, -49.87, -106.48) mm, rotated rx -172.19 ry 6.28 rz 7.52 deg; joints [-6.012, -28.251, 92.717, 91.394, 105.363, 46.294, -36.259]
  MoveL 5078 to (-26.87, -49.26, -106.49) mm, rotated rx -172.19 ry 6.28 rz 7.52 deg; joints [-6.002, -28.224, 92.655, 91.413, 105.357, 46.33, -36.259]
  MoveL 5079 to (-27.27, -48.6, -106.49) mm, rotated rx -172.19 ry 6.28 rz 7.52 deg; joints [-5.988, -28.196, 92.587, 91.437, 105.35, 46.371, -36.259]
  MoveL 5080 to (-27.18, -50.53, -108.04) mm, rotated rx -172.19 ry 6.28 rz 7.52 deg; joints [-6.01, -28.359, 92.781, 91.408, 105.361, 46.339, -36.259]
  MoveL 5081 to (-28.73, -48.75, -108.17) mm, rotated rx -172.19 ry 6.28 rz 7.52 deg; joints [-5.958, -28.296, 92.598, 91.488, 105.335, 46.462, -36.259]
  MoveL 5082 to (-30.19, -47.06, -108.28) mm, rotated rx -172.19 ry 6.28 rz 7.52 deg; joints [-5.908, -28.234, 92.425, 91.564, 105.31, 46.578, -36.259]
  MoveL 5083 to (-31.62, -45.43, -108.44) mm, rotated rx -172.19 ry 6.28 rz 7.52 deg; joints [-5.86, -28.178, 92.258, 91.637, 105.286, 46.692, -36.259]
  MoveL 5084 to (-33.01, -43.82, -108.55) mm, rotated rx -172.19 ry 6.28 rz 7.52 deg; joints [-5.813, -28.119, 92.091, 91.709, 105.263, 46.803, -36.259]
  MoveL 5085 to (-34.41, -42.2, -108.66) mm, rotated rx -172.19 ry 6.28 rz 7.52 deg; joints [-5.765, -28.06, 91.924, 91.78, 105.238, 46.914, -36.259]
  MoveL 5086 to (-35.81, -40.6, -108.88) mm, rotated rx -172.19 ry 6.28 rz 7.52 deg; joints [-5.719, -28.005, 91.757, 91.852, 105.214, 47.031, -36.259]
  MoveL 5087 to (-37.21, -38.98, -109.11) mm, rotated rx -172.19 ry 6.28 rz 7.52 deg; joints [-5.673, -27.951, 91.589, 91.924, 105.19, 47.147, -36.259]
  MoveL 5088 to (-38.6, -37.36, -109.22) mm, rotated rx -172.19 ry 6.28 rz 7.52 deg; joints [-5.627, -27.89, 91.42, 91.995, 105.166, 47.259, -36.259]
  MoveL 5089 to (-39.98, -35.73, -109.22) mm, rotated rx -172.19 ry 6.28 rz 7.52 deg; joints [-5.579, -27.825, 91.25, 92.066, 105.141, 47.366, -36.259]
  MoveL 5090 to (-41.37, -34.11, -109.33) mm, rotated rx -172.19 ry 6.28 rz 7.52 deg; joints [-5.533, -27.764, 91.08, 92.136, 105.116, 47.478, -36.259]
  MoveL 5091 to (-42.77, -32.47, -109.54) mm, rotated rx -172.19 ry 6.28 rz 7.52 deg; joints [-5.487, -27.706, 90.907, 92.208, 105.091, 47.596, -36.259]
  MoveL 5092 to (-44.08, -30.93, -109.72) mm, rotated rx -172.19 ry 6.28 rz 7.52 deg; joints [-5.444, -27.65, 90.745, 92.275, 105.068, 47.706, -36.259]
  MoveL 5093 to (-45.28, -29.52, -109.93) mm, rotated rx -172.19 ry 6.28 rz 7.52 deg; joints [-5.405, -27.601, 90.595, 92.336, 105.046, 47.809, -36.259]
  MoveL 5094 to (-46.55, -28.02, -110.02) mm, rotated rx -172.19 ry 6.28 rz 7.52 deg; joints [-5.363, -27.544, 90.437, 92.401, 105.023, 47.913, -36.259]
  MoveL 5095 to (-47.9, -26.42, -110.04) mm, rotated rx -172.19 ry 6.28 rz 7.52 deg; joints [-5.317, -27.479, 90.268, 92.469, 104.997, 48.019, -36.259]
  MoveL 5096 to (-49.64, -24.34, -110.13) mm, rotated rx -172.19 ry 6.28 rz 7.52 deg; joints [-5.259, -27.396, 90.048, 92.557, 104.965, 48.161, -36.259]
  MoveL 5097 to (-50.94, -22.78, -110.35) mm, rotated rx -172.19 ry 6.28 rz 7.52 deg; joints [-5.217, -27.34, 89.881, 92.624, 104.941, 48.274, -36.259]
  MoveL 5098 to (-52.34, -21.08, -110.55) mm, rotated rx -172.19 ry 6.28 rz 7.52 deg; joints [-5.172, -27.276, 89.699, 92.695, 104.914, 48.396, -36.259]
  MoveL 5099 to (-53.62, -19.51, -110.83) mm, rotated rx -172.19 ry 6.28 rz 7.52 deg; joints [-5.132, -27.221, 89.53, 92.76, 104.89, 48.512, -36.259]
  MoveL 5100 to (-54.89, -17.99, -110.96) mm, rotated rx -172.19 ry 6.28 rz 7.52 deg; joints [-5.091, -27.162, 89.367, 92.824, 104.866, 48.619, -36.259]
  MoveL 5101 to (-56.25, -16.39, -110.98) mm, rotated rx -172.19 ry 6.28 rz 7.52 deg; joints [-5.045, -27.096, 89.195, 92.892, 104.84, 48.727, -36.259]
  MoveL 5102 to (-57.35, -15.01, -111.21) mm, rotated rx -172.19 ry 6.28 rz 7.52 deg; joints [-5.011, -27.045, 89.045, 92.949, 104.818, 48.829, -36.259]
  Set speed (1000.0 mm/s)
  MoveL 5103 to (-80.97, -3.99, -111.21) mm, rotated rx -172.19 ry 6.28 rz 7.52 deg; joints [-4.227, -26.767, 87.82, 93.878, 104.389, 49.782, -36.259]
  Set speed (1000.0 mm/s)
  MoveL 5104 to (-78.2, 1.93, -122.4) mm, rotated rx -172.19 ry 6.28 rz 7.52 deg; joints [-4.45, -26.834, 87.128, 93.881, 104.446, 50.571, -36.259]
  Set speed (100.0 mm/s)
  MoveL 5105 to (-59.92, -6.59, -122.4) mm, rotated rx -172.19 ry 6.28 rz 7.52 deg; joints [-5.054, -27.059, 88.085, 93.168, 104.787, 49.835, -36.259]
  MoveL 5106 to (-58.76, -8.38, -122.4) mm, rotated rx -172.19 ry 6.28 rz 7.52 deg; joints [-5.093, -27.141, 88.279, 93.104, 104.812, 49.72, -36.259]
  MoveL 5107 to (-57.56, -10.26, -122.3) mm, rotated rx -172.19 ry 6.28 rz 7.52 deg; joints [-5.132, -27.224, 88.484, 93.038, 104.837, 49.596, -36.259]
  MoveL 5108 to (-56.33, -12.26, -122.01) mm, rotated rx -172.19 ry 6.28 rz 7.52 deg; joints [-5.17, -27.305, 88.701, 92.969, 104.863, 49.456, -36.259]
  MoveL 5109 to (-55.15, -14.18, -121.66) mm, rotated rx -172.19 ry 6.28 rz 7.52 deg; joints [-5.206, -27.38, 88.91, 92.902, 104.887, 49.319, -36.259]
  MoveL 5110 to (-54.04, -15.93, -121.47) mm, rotated rx -172.19 ry 6.28 rz 7.52 deg; joints [-5.241, -27.452, 89.098, 92.841, 104.909, 49.199, -36.259]
  MoveL 5111 to (-52.99, -17.57, -121.33) mm, rotated rx -172.19 ry 6.28 rz 7.52 deg; joints [-5.275, -27.521, 89.275, 92.782, 104.931, 49.089, -36.259]
  MoveL 5112 to (-51.87, -19.29, -121.28) mm, rotated rx -172.19 ry 6.28 rz 7.52 deg; joints [-5.313, -27.597, 89.46, 92.721, 104.953, 48.978, -36.259]
  MoveL 5113 to (-50.71, -21.08, -121.26) mm, rotated rx -172.19 ry 6.28 rz 7.52 deg; joints [-5.352, -27.677, 89.65, 92.656, 104.977, 48.863, -36.259]
  MoveL 5114 to (-49.55, -22.86, -121.14) mm, rotated rx -172.19 ry 6.28 rz 7.52 deg; joints [-5.39, -27.752, 89.84, 92.592, 105, 48.746, -36.259]
  MoveL 5115 to (-48.31, -24.78, -120.88) mm, rotated rx -172.19 ry 6.28 rz 7.52 deg; joints [-5.43, -27.827, 90.046, 92.523, 105.025, 48.612, -36.259]
  MoveL 5116 to (-46.99, -26.79, -120.7) mm, rotated rx -172.19 ry 6.28 rz 7.52 deg; joints [-5.473, -27.909, 90.259, 92.45, 105.05, 48.477, -36.259]
  MoveL 5117 to (-45.71, -28.74, -120.5) mm, rotated rx -172.19 ry 6.28 rz 7.52 deg; joints [-5.514, -27.988, 90.466, 92.378, 105.075, 48.345, -36.259]
  MoveL 5118 to (-44.54, -30.52, -120.38) mm, rotated rx -172.19 ry 6.28 rz 7.52 deg; joints [-5.553, -28.062, 90.655, 92.313, 105.098, 48.227, -36.259]
  MoveL 5119 to (-42.21, -34.05, -120.11) mm, rotated rx -172.19 ry 6.28 rz 7.52 deg; joints [-5.63, -28.205, 91.026, 92.183, 105.142, 47.993, -36.259]
  MoveL 5120 to (-41.02, -35.87, -120.04) mm, rotated rx -172.19 ry 6.28 rz 7.52 deg; joints [-5.671, -28.282, 91.216, 92.117, 105.165, 47.876, -36.259]
  MoveL 5121 to (-39.83, -37.64, -119.82) mm, rotated rx -172.19 ry 6.28 rz 7.52 deg; joints [-5.71, -28.35, 91.402, 92.05, 105.187, 47.754, -36.259]
  MoveL 5122 to (-38.65, -39.39, -119.66) mm, rotated rx -172.19 ry 6.28 rz 7.52 deg; joints [-5.749, -28.419, 91.585, 91.985, 105.208, 47.637, -36.259]
  MoveL 5123 to (-37.47, -41.14, -119.48) mm, rotated rx -172.19 ry 6.28 rz 7.52 deg; joints [-5.788, -28.486, 91.768, 91.919, 105.23, 47.519, -36.259]
  MoveL 5124 to (-36.26, -42.95, -119.39) mm, rotated rx -172.19 ry 6.28 rz 7.52 deg; joints [-5.829, -28.56, 91.956, 91.851, 105.252, 47.401, -36.259]
  MoveL 5125 to (-34.99, -44.83, -119.26) mm, rotated rx -172.19 ry 6.28 rz 7.52 deg; joints [-5.872, -28.635, 92.151, 91.78, 105.275, 47.277, -36.259]
  MoveL 5126 to (-33.95, -46.43, -119.2) mm, rotated rx -172.19 ry 6.28 rz 7.52 deg; joints [-5.908, -28.701, 92.316, 91.721, 105.294, 47.175, -36.259]
  MoveL 5127 to (-33.39, -46.06, -118.32) mm, rotated rx -172.19 ry 6.28 rz 7.52 deg; joints [-5.916, -28.638, 92.282, 91.706, 105.298, 47.145, -36.259]
  MoveL 5128 to (-33.37, -45.7, -117.9) mm, rotated rx -172.19 ry 6.28 rz 7.52 deg; joints [-5.912, -28.602, 92.247, 91.709, 105.297, 47.144, -36.259]
  MoveL 5129 to (-33.33, -45.65, -117.62) mm, rotated rx -172.19 ry 6.28 rz 7.52 deg; joints [-5.91, -28.587, 92.242, 91.708, 105.296, 47.133, -36.259]
  MoveL 5130 to (-33.28, -45.97, -117.51) mm, rotated rx -172.19 ry 6.28 rz 7.52 deg; joints [-5.91, -28.599, 92.276, 91.702, 105.297, 47.11, -36.259]
  MoveL 5131 to (-33.25, -46.42, -117.44) mm, rotated rx -172.19 ry 6.28 rz 7.52 deg; joints [-5.911, -28.62, 92.323, 91.694, 105.298, 47.083, -36.259]
  MoveL 5132 to (-33.23, -46.98, -117.41) mm, rotated rx -172.19 ry 6.28 rz 7.52 deg; joints [-5.912, -28.648, 92.381, 91.685, 105.299, 47.052, -36.259]
  MoveL 5133 to (-33.22, -47.68, -117.37) mm, rotated rx -172.19 ry 6.28 rz 7.52 deg; joints [-5.912, -28.682, 92.453, 91.674, 105.3, 47.013, -36.259]
  MoveL 5134 to (-33.21, -48.31, -117.35) mm, rotated rx -172.19 ry 6.28 rz 7.52 deg; joints [-5.913, -28.715, 92.519, 91.665, 105.302, 46.979, -36.259]
  MoveL 5135 to (-33.22, -48.84, -117.35) mm, rotated rx -172.19 ry 6.28 rz 7.52 deg; joints [-5.913, -28.742, 92.573, 91.657, 105.302, 46.951, -36.259]
  MoveL 5136 to (-33.21, -49.32, -117.33) mm, rotated rx -172.19 ry 6.28 rz 7.52 deg; joints [-5.913, -28.767, 92.623, 91.65, 105.303, 46.925, -36.259]
  MoveL 5137 to (-33.17, -50.36, -117.25) mm, rotated rx -172.19 ry 6.28 rz 7.52 deg; joints [-5.915, -28.817, 92.731, 91.633, 105.306, 46.866, -36.259]
  MoveL 5138 to (-33.14, -50.92, -117.2) mm, rotated rx -172.19 ry 6.28 rz 7.52 deg; joints [-5.915, -28.845, 92.788, 91.624, 105.307, 46.834, -36.259]
  MoveL 5139 to (-33.1, -51.43, -117.14) mm, rotated rx -172.19 ry 6.28 rz 7.52 deg; joints [-5.916, -28.868, 92.841, 91.615, 105.308, 46.803, -36.259]
  MoveL 5140 to (-33.06, -51.89, -117.06) mm, rotated rx -172.19 ry 6.28 rz 7.52 deg; joints [-5.917, -28.888, 92.889, 91.607, 105.309, 46.775, -36.259]
  MoveL 5141 to (-33.02, -52.36, -117) mm, rotated rx -172.19 ry 6.28 rz 7.52 deg; joints [-5.918, -28.91, 92.937, 91.599, 105.31, 46.748, -36.259]
  MoveL 5142 to (-33.01, -52.84, -116.97) mm, rotated rx -172.19 ry 6.28 rz 7.52 deg; joints [-5.919, -28.933, 92.986, 91.591, 105.311, 46.72, -36.259]
  MoveL 5143 to (-33, -53.36, -116.95) mm, rotated rx -172.19 ry 6.28 rz 7.52 deg; joints [-5.919, -28.96, 93.04, 91.584, 105.312, 46.692, -36.259]
  MoveL 5144 to (-33.04, -57.03, -116.95) mm, rotated rx -172.19 ry 6.28 rz 7.52 deg; joints [-5.92, -29.151, 93.416, 91.532, 105.318, 46.501, -36.259]
  MoveL 5145 to (-33.17, -58.65, -116.97) mm, rotated rx -172.19 ry 6.28 rz 7.52 deg; joints [-5.917, -29.238, 93.582, 91.513, 105.319, 46.42, -36.259]
  MoveL 5146 to (-33.31, -59.21, -117) mm, rotated rx -172.19 ry 6.28 rz 7.52 deg; joints [-5.913, -29.27, 93.639, 91.51, 105.318, 46.394, -36.259]
  MoveL 5147 to (-33.49, -59.61, -117.03) mm, rotated rx -172.19 ry 6.28 rz 7.52 deg; joints [-5.908, -29.296, 93.68, 91.51, 105.316, 46.377, -36.259]
  MoveL 5148 to (-33.7, -59.88, -117.08) mm, rotated rx -172.19 ry 6.28 rz 7.52 deg; joints [-5.901, -29.314, 93.707, 91.514, 105.313, 46.369, -36.259]
  MoveL 5149 to (-33.82, -59.96, -117.1) mm, rotated rx -172.19 ry 6.28 rz 7.52 deg; joints [-5.898, -29.321, 93.715, 91.517, 105.311, 46.367, -36.259]
  MoveL 5150 to (-33.95, -60.01, -117.12) mm, rotated rx -172.19 ry 6.28 rz 7.52 deg; joints [-5.893, -29.327, 93.721, 91.521, 105.31, 46.368, -36.259]
  MoveL 5151 to (-34.09, -60.04, -117.15) mm, rotated rx -172.19 ry 6.28 rz 7.52 deg; joints [-5.889, -29.332, 93.723, 91.525, 105.308, 46.37, -36.259]
  MoveL 5152 to (-34.23, -60.03, -117.18) mm, rotated rx -172.19 ry 6.28 rz 7.52 deg; joints [-5.885, -29.335, 93.722, 91.53, 105.306, 46.373, -36.259]
  MoveL 5153 to (-34.54, -59.95, -117.24) mm, rotated rx -172.19 ry 6.28 rz 7.52 deg; joints [-5.875, -29.337, 93.714, 91.542, 105.301, 46.385, -36.259]
  MoveL 5154 to (-35.2, -59.51, -117.37) mm, rotated rx -172.19 ry 6.28 rz 7.52 deg; joints [-5.853, -29.33, 93.669, 91.572, 105.291, 46.424, -36.259]
  MoveL 5155 to (-35.91, -58.8, -117.51) mm, rotated rx -172.19 ry 6.28 rz 7.52 deg; joints [-5.83, -29.31, 93.596, 91.607, 105.279, 46.478, -36.259]
  MoveL 5156 to (-37.34, -56.94, -117.78) mm, rotated rx -172.19 ry 6.28 rz 7.52 deg; joints [-5.783, -29.246, 93.406, 91.684, 105.255, 46.608, -36.259]
  MoveL 5157 to (-38.68, -54.93, -118.02) mm, rotated rx -172.19 ry 6.28 rz 7.52 deg; joints [-5.739, -29.171, 93.199, 91.76, 105.232, 46.744, -36.259]
  MoveL 5158 to (-68.35, -9.83, -123.1) mm, rotated rx -172.19 ry 6.28 rz 7.52 deg; joints [-4.783, -27.381, 88.419, 93.4, 104.657, 49.815, -36.259]
  MoveL 5159 to (-70.45, -6.63, -123.47) mm, rotated rx -172.19 ry 6.28 rz 7.52 deg; joints [-4.717, -27.247, 88.068, 93.513, 104.612, 50.037, -36.259]
  MoveL 5160 to (-72.36, -3.4, -123.88) mm, rotated rx -172.19 ry 6.28 rz 7.52 deg; joints [-4.659, -27.11, 87.713, 93.62, 104.57, 50.26, -36.259]
  MoveL 5161 to (-72.87, -2, -124.09) mm, rotated rx -172.19 ry 6.28 rz 7.52 deg; joints [-4.645, -27.047, 87.559, 93.656, 104.557, 50.354, -36.259]
  MoveL 5162 to (-72.91, -1.46, -124.19) mm, rotated rx -172.19 ry 6.28 rz 7.52 deg; joints [-4.645, -27.021, 87.499, 93.665, 104.555, 50.388, -36.259]
  MoveL 5163 to (-72.86, -1.23, -124.23) mm, rotated rx -172.19 ry 6.28 rz 7.52 deg; joints [-4.647, -27.009, 87.475, 93.667, 104.555, 50.402, -36.259]
  MoveL 5164 to (-72.76, -1.05, -124.27) mm, rotated rx -172.19 ry 6.28 rz 7.52 deg; joints [-4.651, -26.999, 87.455, 93.666, 104.556, 50.412, -36.259]
  MoveL 5165 to (-72.6, -0.91, -124.31) mm, rotated rx -172.19 ry 6.28 rz 7.52 deg; joints [-4.656, -26.991, 87.44, 93.663, 104.559, 50.419, -36.259]
  MoveL 5166 to (-72.39, -0.82, -124.35) mm, rotated rx -172.19 ry 6.28 rz 7.52 deg; joints [-4.664, -26.984, 87.43, 93.657, 104.562, 50.423, -36.259]
  MoveL 5167 to (-72.12, -0.77, -124.37) mm, rotated rx -172.19 ry 6.28 rz 7.52 deg; joints [-4.673, -26.979, 87.425, 93.649, 104.567, 50.423, -36.259]
  MoveL 5168 to (-71.78, -0.78, -124.4) mm, rotated rx -172.19 ry 6.28 rz 7.52 deg; joints [-4.684, -26.976, 87.426, 93.638, 104.573, 50.418, -36.259]
  MoveL 5169 to (-69.68, -1.41, -124.45) mm, rotated rx -172.19 ry 6.28 rz 7.52 deg; joints [-4.754, -26.985, 87.499, 93.561, 104.611, 50.355, -36.259]
  MoveL 5170 to (-67.75, -2.23, -124.45) mm, rotated rx -172.19 ry 6.28 rz 7.52 deg; joints [-4.818, -27.004, 87.591, 93.487, 104.647, 50.281, -36.259]
  MoveL 5171 to (-64.45, -4.13, -124.49) mm, rotated rx -172.19 ry 6.28 rz 7.52 deg; joints [-4.928, -27.066, 87.802, 93.353, 104.709, 50.131, -36.259]
  MoveL 5172 to (-61.84, -6.53, -124.6) mm, rotated rx -172.19 ry 6.28 rz 7.52 deg; joints [-5.016, -27.167, 88.064, 93.235, 104.761, 49.967, -36.259]
  MoveL 5173 to (-58.52, -11.58, -124.9) mm, rotated rx -172.19 ry 6.28 rz 7.52 deg; joints [-5.131, -27.411, 88.611, 93.055, 104.834, 49.658, -36.259]
  MoveL 5174 to (-57.66, -13.78, -125.03) mm, rotated rx -172.19 ry 6.28 rz 7.52 deg; joints [-5.162, -27.525, 88.847, 92.996, 104.855, 49.532, -36.259]
  MoveL 5175 to (-46.4, -46.68, -126.9) mm, rotated rx -172.19 ry 6.28 rz 7.52 deg; joints [-5.576, -29.21, 92.306, 92.158, 105.127, 47.707, -36.259]
  MoveL 5176 to (-45.42, -49.49, -127.06) mm, rotated rx -172.19 ry 6.28 rz 7.52 deg; joints [-5.612, -29.351, 92.595, 92.085, 105.149, 47.554, -36.259]
  MoveL 5177 to (-43.78, -52.84, -127.3) mm, rotated rx -172.19 ry 6.28 rz 7.52 deg; joints [-5.673, -29.513, 92.939, 91.982, 105.183, 47.367, -36.259]
  MoveL 5178 to (-42.85, -53.99, -127.44) mm, rotated rx -172.19 ry 6.28 rz 7.52 deg; joints [-5.707, -29.565, 93.056, 91.934, 105.201, 47.3, -36.259]
  MoveL 5179 to (-42.39, -54.3, -127.51) mm, rotated rx -172.19 ry 6.28 rz 7.52 deg; joints [-5.724, -29.578, 93.087, 91.914, 105.209, 47.281, -36.259]
  MoveL 5180 to (-42.18, -54.36, -127.55) mm, rotated rx -172.19 ry 6.28 rz 7.52 deg; joints [-5.732, -29.579, 93.094, 91.905, 105.212, 47.276, -36.259]
  MoveL 5181 to (-41.97, -54.37, -127.58) mm, rotated rx -172.19 ry 6.28 rz 7.52 deg; joints [-5.739, -29.578, 93.094, 91.898, 105.216, 47.275, -36.259]
  MoveL 5182 to (-41.77, -54.3, -127.62) mm, rotated rx -172.19 ry 6.28 rz 7.52 deg; joints [-5.746, -29.573, 93.087, 91.892, 105.219, 47.277, -36.259]
  MoveL 5183 to (-41.58, -54.16, -127.65) mm, rotated rx -172.19 ry 6.28 rz 7.52 deg; joints [-5.753, -29.564, 93.073, 91.888, 105.222, 47.283, -36.259]
  MoveL 5184 to (-41.4, -53.95, -127.69) mm, rotated rx -172.19 ry 6.28 rz 7.52 deg; joints [-5.759, -29.551, 93.05, 91.885, 105.224, 47.293, -36.259]
  MoveL 5185 to (-41.24, -53.64, -127.72) mm, rotated rx -172.19 ry 6.28 rz 7.52 deg; joints [-5.765, -29.534, 93.019, 91.884, 105.226, 47.308, -36.259]
  MoveL 5186 to (-40.76, -51.5, -127.84) mm, rotated rx -172.19 ry 6.28 rz 7.52 deg; joints [-5.782, -29.419, 92.798, 91.898, 105.23, 47.417, -36.259]
  MoveL 5187 to (-40.7, -50.99, -127.86) mm, rotated rx -172.19 ry 6.28 rz 7.52 deg; joints [-5.783, -29.392, 92.745, 91.903, 105.23, 47.444, -36.259]
  MoveL 5188 to (-40.68, -50.53, -127.91) mm, rotated rx -172.19 ry 6.28 rz 7.52 deg; joints [-5.785, -29.369, 92.698, 91.909, 105.23, 47.47, -36.259]
  MoveL 5189 to (-40.67, -50.09, -127.98) mm, rotated rx -172.19 ry 6.28 rz 7.52 deg; joints [-5.785, -29.349, 92.652, 91.915, 105.229, 47.496, -36.259]
  MoveL 5190 to (-40.65, -49.65, -128.04) mm, rotated rx -172.19 ry 6.28 rz 7.52 deg; joints [-5.786, -29.328, 92.606, 91.921, 105.229, 47.522, -36.259]
  MoveL 5191 to (-40.62, -49.18, -128.07) mm, rotated rx -172.19 ry 6.28 rz 7.52 deg; joints [-5.788, -29.304, 92.558, 91.926, 105.229, 47.547, -36.259]
  MoveL 5192 to (-39.98, -44.54, -128.08) mm, rotated rx -172.19 ry 6.28 rz 7.52 deg; joints [-5.806, -29.049, 92.078, 91.971, 105.229, 47.78, -36.259]
  MoveL 5193 to (-39.93, -44.1, -128.11) mm, rotated rx -172.19 ry 6.28 rz 7.52 deg; joints [-5.808, -29.026, 92.032, 91.976, 105.229, 47.803, -36.259]
  MoveL 5194 to (-39.87, -43.63, -128.12) mm, rotated rx -172.19 ry 6.28 rz 7.52 deg; joints [-5.81, -29, 91.983, 91.98, 105.229, 47.828, -36.259]
  MoveL 5195 to (-39.73, -42.61, -128.12) mm, rotated rx -172.19 ry 6.28 rz 7.52 deg; joints [-5.814, -28.944, 91.877, 91.99, 105.23, 47.88, -36.259]
  MoveL 5196 to (-39.66, -42.04, -128.13) mm, rotated rx -172.19 ry 6.28 rz 7.52 deg; joints [-5.816, -28.913, 91.818, 91.996, 105.23, 47.909, -36.259]
  MoveL 5197 to (-39.61, -41.44, -128.14) mm, rotated rx -172.19 ry 6.28 rz 7.52 deg; joints [-5.817, -28.881, 91.755, 92.003, 105.229, 47.94, -36.259]
  MoveL 5198 to (-39.59, -40.77, -128.17) mm, rotated rx -172.19 ry 6.28 rz 7.52 deg; joints [-5.818, -28.846, 91.686, 92.012, 105.228, 47.976, -36.259]
  MoveL 5199 to (-39.65, -40.11, -128.2) mm, rotated rx -172.19 ry 6.28 rz 7.52 deg; joints [-5.816, -28.813, 91.617, 92.024, 105.226, 48.013, -36.259]
  MoveL 5200 to (-39.76, -39.47, -128.21) mm, rotated rx -172.19 ry 6.28 rz 7.52 deg; joints [-5.812, -28.781, 91.55, 92.037, 105.223, 48.049, -36.259]
  MoveL 5201 to (-39.83, -40.78, -129.19) mm, rotated rx -172.19 ry 6.28 rz 7.52 deg; joints [-5.822, -28.891, 91.681, 92.022, 105.228, 48.027, -36.259]
  MoveL 5202 to (-40.69, -39.75, -129.62) mm, rotated rx -172.19 ry 6.28 rz 7.52 deg; joints [-5.797, -28.865, 91.572, 92.067, 105.214, 48.114, -36.259]
  MoveL 5203 to (-41.53, -38.52, -129.94) mm, rotated rx -172.19 ry 6.28 rz 7.52 deg; joints [-5.772, -28.825, 91.442, 92.114, 105.199, 48.206, -36.259]
  MoveL 5204 to (-42.39, -37.06, -130.17) mm, rotated rx -172.19 ry 6.28 rz 7.52 deg; joints [-5.744, -28.768, 91.288, 92.164, 105.183, 48.307, -36.259]
  MoveL 5205 to (-43.37, -35.16, -130.39) mm, rotated rx -172.19 ry 6.28 rz 7.52 deg; joints [-5.713, -28.69, 91.088, 92.225, 105.163, 48.431, -36.259]
  MoveL 5206 to (-44.32, -33.25, -130.5) mm, rotated rx -172.19 ry 6.28 rz 7.52 deg; joints [-5.681, -28.606, 90.888, 92.285, 105.144, 48.551, -36.259]
  MoveL 5207 to (-45.27, -31.34, -130.61) mm, rotated rx -172.19 ry 6.28 rz 7.52 deg; joints [-5.649, -28.521, 90.686, 92.344, 105.124, 48.671, -36.259]
  MoveL 5208 to (-46.24, -29.44, -130.84) mm, rotated rx -172.19 ry 6.28 rz 7.52 deg; joints [-5.618, -28.441, 90.484, 92.404, 105.105, 48.797, -36.259]
  MoveL 5209 to (-47.18, -27.52, -130.96) mm, rotated rx -172.19 ry 6.28 rz 7.52 deg; joints [-5.587, -28.356, 90.282, 92.463, 105.085, 48.918, -36.259]
  MoveL 5210 to (-48.13, -25.61, -131.19) mm, rotated rx -172.19 ry 6.28 rz 7.52 deg; joints [-5.556, -28.275, 90.079, 92.523, 105.066, 49.044, -36.259]
  MoveL 5211 to (-49.07, -23.7, -131.31) mm, rotated rx -172.19 ry 6.28 rz 7.52 deg; joints [-5.525, -28.189, 89.875, 92.582, 105.046, 49.165, -36.259]
  MoveL 5212 to (-50.01, -21.78, -131.43) mm, rotated rx -172.19 ry 6.28 rz 7.52 deg; joints [-5.494, -28.103, 89.67, 92.641, 105.026, 49.287, -36.259]
  MoveL 5213 to (-50.95, -19.86, -131.66) mm, rotated rx -172.19 ry 6.28 rz 7.52 deg; joints [-5.465, -28.02, 89.464, 92.699, 105.006, 49.414, -36.259]
  MoveL 5214 to (-51.83, -18.02, -131.77) mm, rotated rx -172.19 ry 6.28 rz 7.52 deg; joints [-5.436, -27.936, 89.267, 92.755, 104.987, 49.53, -36.259]
  MoveL 5215 to (-52.68, -16.23, -131.97) mm, rotated rx -172.19 ry 6.28 rz 7.52 deg; joints [-5.409, -27.858, 89.074, 92.809, 104.968, 49.649, -36.259]
  MoveL 5216 to (-53.73, -14.1, -132.13) mm, rotated rx -172.19 ry 6.28 rz 7.52 deg; joints [-5.375, -27.762, 88.844, 92.874, 104.945, 49.786, -36.259]
  MoveL 5217 to (-54.89, -11.64, -132.22) mm, rotated rx -172.19 ry 6.28 rz 7.52 deg; joints [-5.336, -27.646, 88.579, 92.948, 104.919, 49.939, -36.259]
  MoveL 5218 to (-55.79, -9.77, -132.29) mm, rotated rx -172.19 ry 6.28 rz 7.52 deg; joints [-5.306, -27.558, 88.377, 93.004, 104.898, 50.057, -36.259]
  MoveL 5219 to (-56.63, -8.04, -132.42) mm, rotated rx -172.19 ry 6.28 rz 7.52 deg; joints [-5.28, -27.479, 88.189, 93.056, 104.88, 50.168, -36.259]
  MoveL 5220 to (-57.49, -6.25, -132.52) mm, rotated rx -172.19 ry 6.28 rz 7.52 deg; joints [-5.252, -27.396, 87.994, 93.11, 104.86, 50.283, -36.259]
  MoveL 5221 to (-58.33, -4.49, -132.63) mm, rotated rx -172.19 ry 6.28 rz 7.52 deg; joints [-5.225, -27.314, 87.802, 93.162, 104.841, 50.396, -36.259]
  MoveL 5222 to (-59.22, -2.63, -132.7) mm, rotated rx -172.19 ry 6.28 rz 7.52 deg; joints [-5.195, -27.225, 87.599, 93.218, 104.82, 50.513, -36.259]
  MoveL 5223 to (-60.17, -0.62, -132.8) mm, rotated rx -172.19 ry 6.28 rz 7.52 deg; joints [-5.164, -27.13, 87.379, 93.277, 104.797, 50.641, -36.259]
  MoveL 5224 to (-61.18, 1.57, -133.06) mm, rotated rx -172.19 ry 6.28 rz 7.52 deg; joints [-5.134, -27.031, 87.138, 93.341, 104.774, 50.787, -36.259]
  MoveL 5225 to (-62.56, 3.33, -134.05) mm, rotated rx -172.19 ry 6.28 rz 7.52 deg; joints [-5.099, -26.989, 86.938, 93.412, 104.747, 50.949, -36.259]
